(*bagFeedMasterMotor(modbusInputParameters := BagDeliverMasterMotorModbusInputs, 
                    stepsPerInchSetpoint := Globals.STEPS_PER_INCH_20_DEGREE_BAG_DELIVERY, 
                    reversePolarity := FALSE, 
                    slave := Bag_Delivery_Master_Motor);*)
bagFeedMasterMotor(ptrEIPInputs := ADR(bagDeliveryMotorInputs),
                ptrEIPOutputs := ADR(bagDeliveryMotorOutputs),
                stepsPerInchSetpoint := Globals.STEPS_PER_INCH_20_DEGREE_BAG_DELIVERY,
                //faultHandler := PRG_Bagger.faultHandler,
				reversePolarity := FALSE, 
				defaultCurrentSetpoint := 1150, 
				commFail := Bag_Delivery_EIP_Motor.eState <> IoDrvEthernetIP.AdapterState.RUNNING);
bagFeedMasterMotor.Execute();

bagFeedRearMotor(ptrEIPInputs := ADR(bagRearMotorInputs),
                ptrEIPOutputs := ADR(bagRearMotorOutputs),
                stepsPerInchSetpoint := Globals.STEPS_PER_INCH_20_DEGREE_BAG_DELIVERY,
                //faultHandler := PRG_Bagger.faultHandler,
				reversePolarity := FALSE, 
				defaultCurrentSetpoint := 1150, 
				commFail := Bag_Delivery_Rear_Motor.eState <> IoDrvEthernetIP.AdapterState.RUNNING);
bagFeedRearMotor.Execute();

IF enableONS.Q OR resetONS.Q THEN
    IF _mode = DEVICE_MODES.Manual THEN 
        state := BAG_DELIVERY_STATES.Manual;
    ELSE
        state := BAG_DELIVERY_STATES.Idle;
    END_IF
	_reset := FALSE;
	ClearCommands();
END_IF
jogForwardONS(CLK := jogForwardPB);
jogReverseONS(CLK := jogReversePB);
IF NOT enable THEN
    state := BAG_DELIVERY_STATES.Idle;
END_IF
delay();
_ready := (_mode = DEVICE_MODES.Auto) AND (NOT (state = BAG_DELIVERY_STATES.Fault) OR NOT (state = BAG_DELIVERY_STATES.Idle));

IF tensionFailONS.OSR THEN
	bagTensionFault.Trigger();
END_IF

CASE state OF
    BAG_DELIVERY_STATES.Idle :                     
													IF _mode = DEVICE_MODES.Manual THEN 
														state := BAG_DELIVERY_STATES.Manual;
													ELSIF NOT iBagNotPresent OR Globals.enableDryCycle THEN
														state := BAG_DELIVERY_STATES.Ready;
													ELSIF iBagNotPresent AND (_amFeedToEye OR _amReverseBag) THEN
														state := BAG_DELIVERY_STATES.FeedToEye;
														_amFeedToEye := FALSE;
													END_IF
													IF jogForwardONS.OSR THEN
														bagFeedMasterMotor.MoveDistance(distance := 30, 
                                                                                    acceleration := accelSetpoint, 
                                                                                    deceleration := decelSetpoint, 
                                                                                    velocity := REAL_TO_INT((1 * Globals.VELOCITY_IPS_MULTIPLIER_ELECTRIC)));
														bagFeedRearMotor.MoveDistance(distance := 30, 
                                                                                    acceleration := accelSetpoint, 
                                                                                    deceleration := decelSetpoint, 
                                                                                    velocity := REAL_TO_INT((1 * Globals.VELOCITY_IPS_MULTIPLIER_ELECTRIC)));
													ELSIF jogReverseONS.OSR THEN
														bagFeedMasterMotor.MoveDistance(distance := -30, 
                                                                                    acceleration := accelSetpoint, 
                                                                                    deceleration := decelSetpoint, 
                                                                                    velocity := REAL_TO_INT((1 * Globals.VELOCITY_IPS_MULTIPLIER_ELECTRIC)));
														bagFeedRearMotor.MoveDistance(distance := -30, 
                                                                                    acceleration := accelSetpoint, 
                                                                                    deceleration := decelSetpoint, 
                                                                                    velocity := REAL_TO_INT((1 * Globals.VELOCITY_IPS_MULTIPLIER_ELECTRIC)));
													ELSIF jogForwardONS.OSF OR jogReverseONS.OSF THEN
														bagFeedMasterMotor.Stop();
														bagFeedRearMotor.Stop();
													END_IF
    
	BAG_DELIVERY_STATES.FeedToEye :					//Feed to photoeye if not present
													bagFeedMasterMotor.MoveDistance(distance := feedToPhotoeyeSetpoint, 
                                                                                    acceleration := accelSetpoint, 
                                                                                    deceleration := decelSetpoint, 
                                                                                    velocity := REAL_TO_INT((feedToPhotoeyeSetpoint * Globals.VELOCITY_IPS_MULTIPLIER_ELECTRIC)));
													bagFeedRearMotor.MoveDistance(distance := feedToPhotoeyeSetpoint, 
                                                                                    acceleration := accelSetpoint, 
                                                                                    deceleration := decelSetpoint, 
                                                                                    velocity := REAL_TO_INT((feedToPhotoeyeSetpoint * Globals.VELOCITY_IPS_MULTIPLIER_ELECTRIC)));
													state := BAG_DELIVERY_STATES.FeedingToEye;
													
	BAG_DELIVERY_STATES.FeedingToEye :				// Stop once photoeye seen
													delay.PT := T#3S;
													delay.IN := TRUE;
													IF NOT iBagNotPresent THEN
														bagFeedMasterMotor.Stop();
														bagFeedRearMotor.Stop();
														state := BAG_DELIVERY_STATES.Idle;
														delay.IN := FALSE;
													END_IF
													IF delay.Q THEN
														state := BAG_DELIVERY_STATES.Fault;
														noBagOverEye.Trigger();
														delay.IN := FALSE;
													END_IF
	
    BAG_DELIVERY_STATES.Reverse :                    // Reverse to break perf
                                                    bagFeedMasterMotor.MoveDistance(distance := reverseDistanceSetpoint, 
                                                                                    acceleration := TO_INT((ABS(reverseDistanceSetpoint) * Globals.STEPS_PER_INCH_20_DEGREE_BAG_DELIVERY) *  accelPercent),
                                                                                    deceleration := TO_INT((ABS(reverseDistanceSetpoint) * Globals.STEPS_PER_INCH_20_DEGREE_BAG_DELIVERY) *  decelPercent), 
                                                                                    velocity := REAL_TO_INT((reverseVelocitySetpoint * Globals.VELOCITY_IPS_MULTIPLIER_ELECTRIC)));  
													bagFeedRearMotor.MoveDistance(distance := reverseDistanceSetpoint, 
                                                                                    acceleration := TO_INT((ABS(reverseDistanceSetpoint) * Globals.STEPS_PER_INCH_20_DEGREE_BAG_DELIVERY) *  accelPercent),
                                                                                    deceleration := TO_INT((ABS(reverseDistanceSetpoint) * Globals.STEPS_PER_INCH_20_DEGREE_BAG_DELIVERY) *  decelPercent), 
                                                                                    velocity := REAL_TO_INT((reverseVelocitySetpoint * Globals.VELOCITY_IPS_MULTIPLIER_ELECTRIC)));    
                                                        state := BAG_DELIVERY_STATES.Reversing;
                                                    
                                                    
    BAG_DELIVERY_STATES.Reversing :                    // Back up until we see the trailing edge of the bag
														 IF iBagNotPresent OR Globals.enableDryCycle THEN
															delay.PT := T#10MS;
															delay.IN := TRUE;
															IF delay.Q THEN
																bagFeedMasterMotor.Stop();
																bagFeedRearMotor.Stop();
																delay.IN := FALSE;
																delayForReverseFault.IN := FALSE;
																state := BAG_DELIVERY_STATES.ReverseToPrinthead;
															END_IF
														ELSIF bagFeedMasterMotor.CommandAcknowledged AND NOT iBagNotPresent THEN
															delayForReverseFault.PT := T#3000MS;
															delayForReverseFault.IN := TRUE;
															IF delayForReverseFault.Q THEN
																reverseFault.Trigger();
																bagFeedMasterMotor.Stop();
																bagFeedRearMotor.Stop();
															delayForReverseFault.IN := FALSE;
															state := BAG_DELIVERY_STATES.Fault; 
															END_IF
															
														END_IF
											
                                                  
													
	BAG_DELIVERY_STATES.ReverseToPrinthead :                    // Reverse to print head
                                                    bagFeedMasterMotor.MoveDistance(distance := reverseToPrintHeadSetpoint, 
                                                                                    acceleration := TO_INT((ABS(reverseToPrintHeadSetpoint) * Globals.STEPS_PER_INCH_20_DEGREE_BAG_DELIVERY) *  accelPercent),
                                                                                    deceleration := TO_INT((ABS(reverseToPrintHeadSetpoint) * Globals.STEPS_PER_INCH_20_DEGREE_BAG_DELIVERY) *  decelPercent), 
                                                                                    velocity := REAL_TO_INT((reverseVelocitySetpoint * Globals.VELOCITY_IPS_MULTIPLIER_ELECTRIC))); 
													bagFeedRearMotor.MoveDistance(distance := reverseToPrintHeadSetpoint, 
                                                                                    acceleration := TO_INT((ABS(reverseToPrintHeadSetpoint) * Globals.STEPS_PER_INCH_20_DEGREE_BAG_DELIVERY) *  accelPercent),
                                                                                    deceleration := TO_INT((ABS(reverseToPrintHeadSetpoint) * Globals.STEPS_PER_INCH_20_DEGREE_BAG_DELIVERY) *  decelPercent), 
                                                                                    velocity := REAL_TO_INT((reverseVelocitySetpoint * Globals.VELOCITY_IPS_MULTIPLIER_ELECTRIC)));    
                                                    state := BAG_DELIVERY_STATES.ReversingToPrintHead;
													
	BAG_DELIVERY_STATES.ReversingToPrintHead :                    // Reverse to break perf
                                                   	delay.PT := T#50MS;
													delay.IN := TRUE;
													
													IF delay.Q THEN
														IF bagFeedMasterMotor.CommandAcknowledged AND bagFeedMasterMotor.InPosition THEN
                                                        	state := BAG_DELIVERY_STATES.ReverseDone;
                                                    	END_IF
														delay.IN := FALSE;
													END_IF
                                                    
    BAG_DELIVERY_STATES.ReverseDone :                // We don't print in semi auto or manual mode.  In auto mode if the printer is selected then we move to those states
                                                    IF _mode = DEVICE_MODES.SemiAuto OR _mode = DEVICE_MODES.Manual OR (_mode  = DEVICE_MODES.Auto AND autoFeedDelay.Q) THEN
                                                        IF bagFeedMasterMotor.CommandAcknowledged THEN
															state := BAG_DELIVERY_STATES.FeedBagOut;
                                                        	remainingLength := bagLengthSetpoint;
                                                        	_amFeedBagOut := FALSE;
														END_IF
														
                                                    ELSIF (_mode  = DEVICE_MODES.Auto AND _amWaitForPrinter) THEN
                                                        IF bagFeedMasterMotor.CommandAcknowledged THEN
															state := BAG_DELIVERY_STATES.WaitingForPrinter;
															remainingLength := bagLengthSetpoint - (printLengthSetpoint + printOffsetSetpoint + printerExtraFeedLength);
															_amWaitForPrinter := FALSE;  
														END_IF  
                                                    END_IF
                                                        
                                                    
    BAG_DELIVERY_STATES.WaitingForPrinter :            // 
                                                    IF (_mode  = DEVICE_MODES.Auto AND _amPrinterReady) THEN
														IF printOffsetSetpoint <> 0 THEN
															state := BAG_DELIVERY_STATES.FeedToPrintOffset;
														ELSE
															state := BAG_DELIVERY_STATES.FedToPrintOffset;
														END_IF
                                                        
                                                        _amPrinterReady := FALSE;
                                                    END_IF
                                                        
    BAG_DELIVERY_STATES.FeedToPrintOffset :            // 
                                                    bagFeedMasterMotor.MoveDistance(distance := printOffsetSetpoint, 
                                                                                    acceleration := accelSetpoint, 
                                                                                    deceleration := decelSetpoint, 
                                                                                    velocity := REAL_TO_INT((feedVelocitySetpoint * Globals.VELOCITY_IPS_MULTIPLIER_ELECTRIC)));  
													bagFeedRearMotor.MoveDistance(distance := printOffsetSetpoint, 
                                                                                    acceleration := accelSetpoint, 
                                                                                    deceleration := decelSetpoint, 
                                                                                    velocity := REAL_TO_INT((feedVelocitySetpoint * Globals.VELOCITY_IPS_MULTIPLIER_ELECTRIC)));  
                                                        state := BAG_DELIVERY_STATES.FeedingToPrintOffset;
                                                    
    BAG_DELIVERY_STATES.FeedingToPrintOffset :        // 
													delay.PT := T#50MS;
													delay.IN := TRUE;
													
													IF delay.Q THEN
														IF bagFeedMasterMotor.CommandAcknowledged AND bagFeedMasterMotor.InPosition THEN
                                                        	state := BAG_DELIVERY_STATES.FedToPrintOffset;
                                                    	END_IF
														delay.IN := FALSE;
													END_IF
                                                    
                                                    
    BAG_DELIVERY_STATES.FedToPrintOffset :            // 
                                                    IF (_mode  = DEVICE_MODES.Auto AND _amStartPrint) THEN
                                                        state := BAG_DELIVERY_STATES.FeedAtPrintSpeed;
                                                        _amStartPrint := FALSE;
                                                    END_IF
                                                    
    BAG_DELIVERY_STATES.FeedAtPrintSpeed :            // 
													delay.PT := delayForPrintFeed;
                                                    delay.IN := TRUE;
													
													IF delay.Q THEN
														bagFeedMasterMotor.MoveDistance(distance := printLengthSetpoint + printerExtraFeedLength, 
                                                                                    acceleration := accelSetpoint, 
                                                                                    deceleration := decelSetpoint, 
                                                                                    velocity := REAL_TO_INT((printVelocitySetpoint * Globals.VELOCITY_IPS_MULTIPLIER_ELECTRIC)));  
														bagFeedRearMotor.MoveDistance(distance := printLengthSetpoint + printerExtraFeedLength, 
                                                                                    acceleration := accelSetpoint, 
                                                                                    deceleration := decelSetpoint, 
                                                                                    velocity := REAL_TO_INT((printVelocitySetpoint * Globals.VELOCITY_IPS_MULTIPLIER_ELECTRIC)));  
                                                        state := BAG_DELIVERY_STATES.FeedingAtPrintSpeed;
														delay.IN := FALSE;
													END_IF
                                                    
    BAG_DELIVERY_STATES.FeedingAtPrintSpeed :        // 
													delay.PT := T#50MS;
													delay.IN := TRUE;
													IF delay.Q THEN
														IF bagFeedMasterMotor.CommandAcknowledged AND bagFeedMasterMotor.InPosition THEN
                                                        	state := BAG_DELIVERY_STATES.FedAtPrintSpeed;
                                                    	END_IF
														delay.IN := FALSE;
													END_IF
                                                   
                                                    
    BAG_DELIVERY_STATES.FedAtPrintSpeed :            // 
                                                    IF (_mode  = DEVICE_MODES.Auto AND _amPrinterDone) THEN
                                                        state := BAG_DELIVERY_STATES.FeedBagOut;
                                                        _amPrinterDone := FALSE;
                                                    END_IF
                                                    
    BAG_DELIVERY_STATES.FeedBagOut :                // Feed bag length out
                                                    //bagFeedMasterMotor.MoveDistanceFinal(distance := (remainingLength + sealOffsetSetpoint + (reverseToPrintHeadSetpoint*-1)), 
													bagFeedMasterMotor.MoveDistanceFinal(distance := (remainingLength + sealBarToPrintHeadLength) - sealOffsetSetpoint, 
                                                                                        acceleration := accelSetpoint, 
                                                                                        deceleration := decelSetpoint, 
                                                                                        velocity := REAL_TO_INT((feedVelocitySetpoint * Globals.VELOCITY_IPS_MULTIPLIER_ELECTRIC)));
													bagFeedRearMotor.MoveDistance(distance := (remainingLength + sealBarToPrintHeadLength) - sealOffsetSetpoint, 
                                                                                        acceleration := accelSetpoint, 
                                                                                        deceleration := decelSetpoint, 
                                                                                        velocity := REAL_TO_INT((feedVelocitySetpoint * Globals.VELOCITY_IPS_MULTIPLIER_ELECTRIC)));
                                                    state := BAG_DELIVERY_STATES.FeedingBagOut;    
    
    BAG_DELIVERY_STATES.FeedingBagOut :                // Wait until move is done
													delay.PT := T#50MS;
													delay.IN := TRUE;
													IF delay.Q THEN
														IF bagFeedMasterMotor.CommandAcknowledged AND bagFeedMasterMotor.InPosition THEN
                                                        state := BAG_DELIVERY_STATES.FedBagOut;
														
                                                    	END_IF
														delay.IN := FALSE;
													END_IF
                                                    
    
    BAG_DELIVERY_STATES.FedBagOut :                    // Go to the next ready state
                                                    IF _mode = DEVICE_MODES.Manual THEN 
                                                        state := BAG_DELIVERY_STATES.Manual;
                                                    ELSE
                                                        state := BAG_DELIVERY_STATES.Ready;
                                                    END_IF
													HMIData.driveRollerClean.SetCount(HMIData.driveRollerClean.count + TO_INT(bagLengthSetpoint));
                                                    Globals.bagDeliveryCycleCount := Globals.bagDeliveryCycleCount + 1;
    
    BAG_DELIVERY_STATES.Ready :                        IF (_mode = DEVICE_MODES.Auto AND _amReverseBag) OR _mode = DEVICE_MODES.SemiAuto THEN 
                                                        state := BAG_DELIVERY_STATES.Reverse;
                                                        ClearCommands();
                                                    END_IF 
													_amFeedToEye := FALSE;
													IF iBagNotPresent AND NOT Globals.enableDryCycle THEN 
														state := BAG_DELIVERY_STATES.Idle;
													END_IF
													IF jogForwardONS.OSR THEN
														bagFeedMasterMotor.MoveDistance(distance := 30, 
                                                                                    acceleration := accelSetpoint, 
                                                                                    deceleration := decelSetpoint, 
                                                                                    velocity := REAL_TO_INT((1 * Globals.VELOCITY_IPS_MULTIPLIER_ELECTRIC)));
														bagFeedRearMotor.MoveDistance(distance := 30, 
                                                                                    acceleration := accelSetpoint, 
                                                                                    deceleration := decelSetpoint, 
                                                                                    velocity := REAL_TO_INT((1 * Globals.VELOCITY_IPS_MULTIPLIER_ELECTRIC)));
													ELSIF jogReverseONS.OSR THEN
														bagFeedMasterMotor.MoveDistance(distance := -30, 
                                                                                    acceleration := accelSetpoint, 
                                                                                    deceleration := decelSetpoint, 
                                                                                    velocity := REAL_TO_INT((1 * Globals.VELOCITY_IPS_MULTIPLIER_ELECTRIC)));
														bagFeedRearMotor.MoveDistance(distance := -30, 
                                                                                    acceleration := accelSetpoint, 
                                                                                    deceleration := decelSetpoint, 
                                                                                    velocity := REAL_TO_INT((1 * Globals.VELOCITY_IPS_MULTIPLIER_ELECTRIC)));
													ELSIF jogForwardONS.OSF OR jogReverseONS.OSF THEN
														bagFeedMasterMotor.Stop();
														bagFeedRearMotor.Stop();
													END_IF
    
    BAG_DELIVERY_STATES.Fault :                        ClearCommands();
													IF jogForwardONS.OSR THEN
														bagFeedMasterMotor.MoveDistance(distance := 30, 
                                                                                    acceleration := accelSetpoint, 
                                                                                    deceleration := decelSetpoint, 
                                                                                    velocity := REAL_TO_INT((1 * Globals.VELOCITY_IPS_MULTIPLIER_ELECTRIC)));
													ELSIF jogReverseONS.OSR THEN
														bagFeedMasterMotor.MoveDistance(distance := -30, 
                                                                                    acceleration := accelSetpoint, 
                                                                                    deceleration := decelSetpoint, 
                                                                                    velocity := REAL_TO_INT((1 * Globals.VELOCITY_IPS_MULTIPLIER_ELECTRIC)));
													ELSIF jogForwardONS.OSF OR jogReverseONS.OSF THEN
														bagFeedMasterMotor.Stop();
														bagFeedRearMotor.Stop();
													END_IF
    
    BAG_DELIVERY_STATES.Manual :                    IF _mode = DEVICE_MODES.Auto THEN
														state := BAG_DELIVERY_STATES.Ready;	
													END_IF
													// Manually feed bags out
                                                    IF feedBagPB THEN
                                                        state := BAG_DELIVERY_STATES.Reverse;
                                                        feedBagPB := FALSE;
                                                    END_IF
                                                        
END_CASE

END_FUNCTION_BLOCK

// FBs/Unused/ElectricPressureBarFB
FUNCTION_BLOCK ElectricPressureBarFB IMPLEMENTS IComponentStatus
VAR_INPUT
    enable : BOOL;
END_VAR
VAR_IN_OUT

END_VAR
VAR_OUTPUT
END_VAR
VAR
    electricPressureBarMotor : FB_FestoMotor();
    delay: TON := (PT := T#1S);
    state : PRESSURE_BAR_STATES;
    enableElectricPressureBarONS : R_TRIG();
    
    _mode : DEVICE_MODES;    // Auto-SemiAuto-Manual
    _ready : BOOL;            // Ready to be controlled
    _amOpenJaw : BOOL;    // Auto Mode Open Jaw Command
    _amCloseJaw : BOOL;     // Auto Mode Close Jaw Command
END_VAR

//    Function Block: ElectricPressureBarFB
//    Description: This function block is the state machine for the electric pressure bar
//    
//    Created by: Ben Hess
//    Created Date: Monday, April 16, 2018

electricPressureBarMotor(deviceType := FML.CMMP_AS,
                                        isFPCActive := TRUE, 
                                        ptrReadFHPPRegister := ADR(%IW145), 
                                        ptrReadFPCRegister := ADR(%IW149),
                                        ptrWriteFHPPRegister := ADR(%QW82),
                                        ptrWriteFPCRegister := ADR(%QW86));                                    
electricPressureBarMotor.Execute();

delay();

//Report as ready if mode is auto and we're not faulted
_ready := (_mode = DEVICE_MODES.Auto) AND NOT (state = PRESSURE_BAR_STATES.Fault);


enableElectricPressureBarONS(CLK := enable);
IF enableElectricPressureBarONS.Q THEN
    state := PRESSURE_BAR_STATES.Idle;
END_IF

IF NOT enable THEN
        state := PRESSURE_BAR_STATES.Fault;
END_IF

CASE state OF
    PRESSURE_BAR_STATES.Idle:        IF enable AND _mode = DEVICE_MODES.SemiAuto OR (_mode = DEVICE_MODES.Auto AND _amCloseJaw) THEN
                                        state := PRESSURE_BAR_STATES.CloseJaw;
                                        _amCloseJaw := FALSE;
                                    END_IF
    
    PRESSURE_BAR_STATES.OpenJaw:    electricPressureBarMotor.ExecuteStoredProgram(1);
                                    IF electricPressureBarMotor.CommandAcknowledged THEN
                                        state := PRESSURE_BAR_STATES.OpeningJaw;
                                        Globals.electricPressureBarCount := Globals.electricPressureBarCount + 1;
                                    END_IF
        
    
    PRESSURE_BAR_STATES.OpeningJaw:    
                                    IF electricPressureBarMotor.ActiveStoredProgramNumber = 1 AND electricPressureBarMotor.InPosition THEN
                                        state := PRESSURE_BAR_STATES.JawOpened;
                                    END_IF
                                    
    PRESSURE_BAR_STATES.JawOpened:     IF _mode = DEVICE_MODES.SemiAuto THEN
                                        delay.IN := TRUE;
                                        IF delay.Q THEN
                                            state := PRESSURE_BAR_STATES.CloseJaw;
                                            delay.IN := FALSE;
                                        END_IF
                                    ELSIF _mode = DEVICE_MODES.Auto AND _amCloseJaw THEN
                                        state := PRESSURE_BAR_STATES.CloseJaw;
                                        _amCloseJaw := FALSE;
                                    END_IF
        
    PRESSURE_BAR_STATES.CloseJaw:    electricPressureBarMotor.ExecuteStoredProgram(2);
                                    IF electricPressureBarMotor.CommandAcknowledged THEN
                                        state := PRESSURE_BAR_STATES.ClosingJaw;
                                        Globals.electricPressureBarCount := Globals.electricPressureBarCount + 1;
                                    END_IF
                                    
    
    PRESSURE_BAR_STATES.ClosingJaw:    IF electricPressureBarMotor.ActiveStoredProgramNumber = 2 AND electricPressureBarMotor.InPosition THEN
                                        state := PRESSURE_BAR_STATES.JawClosed;
                                    END_IF
                                    
    PRESSURE_BAR_STATES.JawClosed:    IF _mode = DEVICE_MODES.SemiAuto THEN
                                        delay.IN := TRUE;
                                        IF delay.Q THEN
                                            state := PRESSURE_BAR_STATES.OpenJaw;
                                            delay.IN := FALSE;
                                        END_IF
                                    ELSIF _mode = DEVICE_MODES.Auto AND _amOpenJaw THEN
                                        state := PRESSURE_BAR_STATES.OpenJaw;
                                        _amOpenJaw := FALSE;
                                    END_IF
    
    PRESSURE_BAR_STATES.Fault:        ClearCommands();        
    
    
END_CASE

END_FUNCTION_BLOCK

// FBs/Unused/MotorizedSealFlattenersFB
FUNCTION_BLOCK MotorizedSealFlattenersFB EXTENDS BaseComponentFB IMPLEMENTS IComponentStatus
VAR_INPUT
    {warning 'TODO: Make a struct for some of these - too many inputs'}
	sealFlattenersVerticalAxis : ICylinder();
    clearanceOffset : REAL := 0.75;        // Clearance Offset in inches
    inSetpoint : REAL := 1.25;            // In setpoint in inches
    outSetpoint : REAL := 17.7;            // Out (sealing) setpoint in inches
    bagHoldingSetpoint : REAL := 17;    // Bag holding setpoint in inches            
    clearanceSpeed : INT := 3000;        // Speed to move in clearance move
    moveInSpeed : INT := 3000;            // Speed to move in in move
    moveOutSpeed : INT := 1000;            // Speed to move in out move
    moveBagHoldingSpeed : INT := 10000;    // Speed to move in bag holding move
    fingersUpSetpoint : REAL := 0;     // Fingers Up setpoint in inches
    fingersDownSetpoint : REAL := 1.1; // Fingers down setpoint in inches
    moveFingersSpeed : INT := 2000;        // Speed to move fingers
    horizontalAxisAccel : INT := 1000;    // Accel setpoint for horizontal axis
    horizontalAxisDecel : INT := 1000;    // Decel Setpoint for horizontal axis
    verticalAxisAccel : INT := 150;    // Accel setpoint for vertical axis
    verticalAxisDecel : INT := 150;    // Decel Setpoint for vertical axis
    testMovePB : BOOL;
    testMoveSP : REAL;
    stopPB : BOOL;
    startPB : BOOL;
    nextSeqPB : BOOL;
    delay : TON := (PT:= T#300MS);
	fingersDownDelay : Standard.TON := (PT := T#200MS);
	
	manualPosSetpoint : REAL;
	
END_VAR
VAR_IN_OUT
	jogIn : BOOL;
	jogOut : BOOL;
	raiseService : BOOL;
	lowerService : BOOL;
	moveToManualSetpoint : BOOL;
END_VAR
VAR_OUTPUT
    state : SEAL_FLATTENER_STATES;
END_VAR
VAR
    //pressureBarMotor : FB_FestoMotor();
    //sealFlattenersVerticalAxisMotor : FB_AppliedMotionStepServoRTU();
	jogInONS: FB_ONS;
	jogOutONS: FB_ONS;
	jogSpeed : INT := 100;
    sealFlattenersHorizontalAxisMotor : FB_AppliedMotionStepServoEIPBaseQX();
	defaultCurrentMSF : DINT := 150;
	outCurrentMSF : DINT := 150;
	bagHoldingCurrentMSF : DINT := 85;
    enableMotorizedSealFlattenersONS : R_TRIG();    
    _amMoveOut : BOOL;                // Auto mode move out command
	_amMoveIn : BOOL;
    _amMoveClearance : BOOL;            // Auto mode move Clearance command
    _amMoveInToBagHolding : BOOL;    // Auto mode move in then bag holding command
END_VAR

//    Function Block:  MotorizedSealFlattenersFB
//    Description: State machine and motor management for motorized seal flateners
//    Currently, this code requires one to use the Oriental drive with pre-programmed 
//    sequence for the horizontal axis
//    Created by: Ben Hess
//    Created Date: Friday, April 6, 2018
SUPER^();
// Setup and execute 2 motor axis'

// Temporary delay between states for testing
fingersDownDelay();
delay();
jogInONS(CLK := jogIn);
jogOutONS(CLK := jogOut);
IF autoModeSelected THEN
    delay.PT := T#300MS;
ELSE
    delay.PT := T#750MS;
END_IF

outSetpoint := HMIData.bagWidth + 0.2;
bagHoldingSetpoint := HMIData.bagWidth;

// Setup the vertical axis motor
sealFlattenersVerticalAxis.Execute();

// Setup the horizontal axis motor 
(*
sealFlattenersHorizontalAxisMotor(modbusInBuffer := OrientalMotorModbusRead,
                stepsPerInchSetpoint := 125,
                reversePolarity := FALSE,
                operatingCurrentDefault := 500,
                modbusCommandOutBuffer := OrientalMotorCommandWrites,
                modbusParametersOutBuffer := OrientalMotorParameterWrites,
                triggerCommandWrite => OrientalMotorTriggerCommandWrite,
                triggerParameterWrite => OrientalMotorTriggerParameterWrite);                
sealFlattenersHorizontalAxisMotor.Execute();
*)

sealFlattenersHorizontalAxisMotor(ptrEIPInputs := ADR(sealFlattenerHorizontalMotorInputs),
                ptrEIPOutputs := ADR(sealFlattenerHorizontalMotorOutputs),
                stepsPerInchSetpoint := Globals.STEPS_PER_INCH_SEAL_FLATTENER_HORIZONTAL_AXIS_MOTOR,
                faultHandler := PRG_Bagger.faultHandler,
				reversePolarity := TRUE, 
				defaultCurrentSetpoint := defaultCurrentMSF, 
				commFail := MSFMotor.eState <> IoDrvEthernetIP.AdapterState.RUNNING,
				isHomable := TRUE);
				
sealFlattenersHorizontalAxisMotor.Execute();

//Report as ready if mode is auto and we're not faulted
_ready := (_mode = DEVICE_MODES.Auto) AND NOT (state = SEAL_FLATTENER_STATES.Fault);

enableMotorizedSealFlattenersONS(CLK := enable);
IF stopPB THEN
    sealFlattenersHorizontalAxisMotor.Stop();
    stopPB := FALSE;
END_IF

IF startPB AND semiAutoModeSelected THEN 
    //sealFlattenersHorizontalAxisMotor.StartOperation();
    startPB := FALSE;
END_IF

IF nextSeqPB THEN 
    //sealFlattenersHorizontalAxisMotor.NextSequence();
    nextSeqPB := FALSE;
END_IF

IF testMovePB THEN
    sealFlattenersHorizontalAxisMotor.MoveToPosition(position := (testMoveSP), acceleration := 100, deceleration := 100, velocity := 600);
    testMovePB := FALSE;
END_IF

IF enableONS.Q OR resetONS.Q THEN 
    state := SEAL_FLATTENER_STATES.Idle;
	sealFlattenersHorizontalAxisMotor.Reset();
	_reset := FALSE;
	ClearCommands();
END_IF

IF NOT enable THEN
    state := SEAL_FLATTENER_STATES.Fault;
END_IF

// State amchine for motorized seal flatteners
CASE state OF
    

    SEAL_FLATTENER_STATES.Idle :                                    //If enabled move to out
                                                                    IF enable AND semiAutoModeSelected OR (autoModeSelected AND _amMoveOut) THEN
                                                                        state := SEAL_FLATTENER_STATES.MoveFlattenersOut;
                                                                        ClearCommands();
                                                                    END_IF
																	
																	IF enable AND autoModeSelected AND _amMoveIn OR _amMoveInToBagHolding THEN
																	//IF enable AND autoModeSelected AND _amMoveIn THEN
																		sealFlattenersVerticalAxis.Retract();
																		state := SEAL_FLATTENER_STATES.MoveFlattenersIn;
																		ClearCommands();
																	END_IF
																	
																	IF jogInONS.OSR THEN
																		sealFlattenersHorizontalAxisMotor.MoveDistance(distance := -18, 
																									acceleration := horizontalAxisAccel, 
																									deceleration := horizontalAxisDecel, 
																									velocity := jogSpeed);
																	ELSIF jogOutONS.OSR THEN
																		sealFlattenersHorizontalAxisMotor.MoveDistance(distance := 18, 
																									acceleration := horizontalAxisAccel, 
																									deceleration := horizontalAxisDecel, 
																									velocity := jogSpeed);
																	ELSIF jogInONS.OSF OR jogOutONS.OSF THEN
																		sealFlattenersHorizontalAxisMotor.Stop();
																	END_IF
																	
																	IF raiseService THEN
																		sealFlattenersVerticalAxis.Retract();  
																		raiseService := FALSE;
																	ELSIF lowerService THEN
																		sealFlattenersVerticalAxis.Extend();  
																		lowerService := FALSE;
																	END_IF
																	
																	IF moveToManualSetpoint THEN
																		sealFlattenersHorizontalAxisMotor.MoveToPosition(position := manualPosSetpoint, 
																									acceleration := horizontalAxisAccel, 
																									deceleration := horizontalAxisDecel, 
																									velocity := moveFingersSpeed);
																		moveToManualSetpoint := FALSE;
																	END_IF
																	
                                                                    
    SEAL_FLATTENER_STATES.MoveFlattenersOut :                        // Move flatteners to out position
                                                                
                                                                    //sealFlattenersHorizontalAxisMotor.StartOperation();
                                                                    sealFlattenersHorizontalAxisMotor.MoveToPositionTorque(position := outSetpoint, 
                                                                                                                        acceleration := horizontalAxisAccel,
                                                                                                                        deceleration := horizontalAxisDecel,
                                                                                                                        velocity := moveOutSpeed,
																														current := outCurrentMSF);                                                    
                                                                    state := SEAL_FLATTENER_STATES.MovingFlattenersOut;
                                                                    
                                                                    
    SEAL_FLATTENER_STATES.MovingFlattenersOut :                        // 
                                                                    delay.IN := TRUE;
                                                                    IF delay.Q THEN
																		IF sealFlattenersHorizontalAxisMotor.CommandAcknowledged AND sealFlattenersHorizontalAxisMotor.CurrentPosition >= (bagHoldingSetpoint - 1.5) THEN
																			state := SEAL_FLATTENER_STATES.MovedFlattenersOut;
                                                                        	delay.IN := FALSE; 
																		END_IF
                                                                    END_IF
                                                                    
    SEAL_FLATTENER_STATES.MovedFlattenersOut :                        // Move flatteners to clearance position state
                                                                    IF enable AND semiAutoModeSelected OR (autoModeSelected AND _amMoveClearance) THEN
                                                                        state := SEAL_FLATTENER_STATES.MoveFlattenersUpAndToClearance;
                                                                        ClearCommands();
                                                                    END_IF
    
    
    SEAL_FLATTENER_STATES.MoveFlattenersUpAndToClearance :                // Move flatteners to clearance position
                                                                    
                                                                    //sealFlattenersHorizontalAxisMotor.NextSequence();
                                                                    sealFlattenersHorizontalAxisMotor.MoveToPosition(position := (outSetpoint - clearanceOffset), 
                                                                                                                        acceleration := horizontalAxisAccel,
                                                                                                                        deceleration := horizontalAxisDecel,
                                                                                                                        velocity := moveOutSpeed);    
                                                                   	sealFlattenersVerticalAxis.Retract();                                                       
                                                                    state := SEAL_FLATTENER_STATES.MovingFlattenersUpAndToClearance;    
    
    
    
    SEAL_FLATTENER_STATES.MovingFlattenersUpAndToClearance :        delay.IN := TRUE;
                                                                    IF delay.Q THEN
																		IF sealFlattenersHorizontalAxisMotor.CommandAcknowledged AND sealFlattenersHorizontalAxisMotor.InPosition THEN
																			state := SEAL_FLATTENER_STATES.MovedFlattenersUpAndToClearance;    
                                                                        	delay.IN := FALSE;
																		END_IF
                                                                    END_IF
                                                                    
                                                                    
    SEAL_FLATTENER_STATES.MovedFlattenersUpAndToClearance :                // Move flatteners to up state
                                                                    IF enable AND semiAutoModeSelected OR (autoModeSelected AND (_amMoveInToBagHolding OR _amMoveIn)) THEN
                                                                        state := SEAL_FLATTENER_STATES.MoveFlattenersIn;
                                                                        //ClearCommands();
                                                                    END_IF
                                        
                                                                    
    SEAL_FLATTENER_STATES.MoveFlattenersIn :                        // Move flatteners up and in
                                                                    //sealFlattenersHorizontalAxisMotor.NextSequence();    
                                                                    sealFlattenersHorizontalAxisMotor.MoveToPosition(position := inSetpoint, 
                                                                                                                        acceleration := horizontalAxisAccel,
                                                                                                                        deceleration := horizontalAxisDecel,
                                                                                                                        velocity := moveInSpeed);                                                    
                                                                    state := SEAL_FLATTENER_STATES.MovingFlattenersIn;
                                                                    
                                                                    
    SEAL_FLATTENER_STATES.MovingFlattenersIn :                        // If we did that command well move on 
                                                                        delay.IN := TRUE;
                                                                        IF delay.Q THEN
																			IF sealFlattenersHorizontalAxisMotor.CommandAcknowledged AND sealFlattenersHorizontalAxisMotor.InPosition THEN
																				state := SEAL_FLATTENER_STATES.MovedFlattenersIn;
                                                                           		delay.IN := FALSE;    
																			END_IF
                                                                        END_IF 
                                                                    
    SEAL_FLATTENER_STATES.MovedFlattenersIn :                        // Now that we're up and in move to down and 4 corners/bag holding
                                                                    IF enable AND semiAutoModeSelected OR (autoModeSelected AND _amMoveInToBagHolding) THEN
                                                                        state := SEAL_FLATTENER_STATES.MoveFlattenersDown;
                                                                        ClearCommands();
                                                                    END_IF    
    
    SEAL_FLATTENER_STATES.MoveFlattenersDown :            // Do moves for down and bag holding
                                                                        
                                                                        sealFlattenersVerticalAxis.Extend();
                                                                                                                                                                                
                                                                        state := SEAL_FLATTENER_STATES.MovingFlattenersDown;
                                                                        
    SEAL_FLATTENER_STATES.MovingFlattenersDown :            
                                                                        //IF sealFlattenersVerticalAxis.CommandAcknowledged AND sealFlattenersVerticalAxis.InPosition THEN
                                                                       	fingersDownDelay.IN := TRUE;
																	  	IF fingersDownDelay.Q THEN
																			state := SEAL_FLATTENER_STATES.MovedFlattenersDown;
																			fingersDownDelay.IN := FALSE;
																		END_IF 
																		
                                                                        //END_IF 
                                                                        
    SEAL_FLATTENER_STATES.MovedFlattenersDown :            state := SEAL_FLATTENER_STATES.MoveFlattenersToBagHolding;
                                                                    
                                                                    
    SEAL_FLATTENER_STATES.MoveFlattenersToBagHolding :            // Do moves for down and bag holding
                                                                        //sealFlattenersHorizontalAxisMotor.NextSequence();    
                                                                        sealFlattenersHorizontalAxisMotor.MoveToPositionTorque(position := bagHoldingSetpoint, 
                                                                                                                        acceleration := horizontalAxisAccel,
                                                                                                                        deceleration := horizontalAxisDecel,
                                                                                                                        velocity := moveBagHoldingSpeed,
																														current := bagHoldingCurrentMSF);                                                
                                                                        state := SEAL_FLATTENER_STATES.MovingFlattenersToBagHolding;
                                                                        
    SEAL_FLATTENER_STATES.MovingFlattenersToBagHolding :            delay.IN := TRUE;
                                                                        IF delay.Q THEN
																			IF sealFlattenersHorizontalAxisMotor.CommandAcknowledged THEN
																				state := SEAL_FLATTENER_STATES.MovedFlattenersToBagHolding;
                                                                            	delay.IN := FALSE; 
																			END_IF   
                                                                        END_IF 
                                                                        
    SEAL_FLATTENER_STATES.MovedFlattenersToBagHolding :            state := SEAL_FLATTENER_STATES.Idle;
																		HMIData.motorizedSealFlattenerCycles.Increment();
                                                                        Globals.motorizedSealFlattenersCount := Globals.motorizedSealFlattenersCount +1;
                                                                        Globals.sealFlattenerFingersCount := Globals.sealFlattenerFingersCount +1;
    SEAL_FLATTENER_STATES.Ready :
    SEAL_FLATTENER_STATES.Fault :
END_CASE

END_FUNCTION_BLOCK

// FBs/Unused/PickAndPlaceFB
FUNCTION_BLOCK PickAndPlaceFB EXTENDS BaseComponentFB
VAR_INPUT
	XAxisMotor : IPositionableMotor;	// X Axis Motor
	YAxisMotor : IPositionableMotor;	// Y Axis Motor
	ZAxisMotor : IPositionableMotor;	// Z Axis Motor
END_VAR
VAR_OUTPUT
	state : VACUUM_PICKER_STATES;	 //State indication
END_VAR
VAR
	
	accel : INT := 2000;
	decel : INT := 2000;
	velo : INT := 2000;
	zVelo : INT := 12000;
END_VAR

//	Function Block: PickAndPlaceFB
//	Description: This provides the methods and state machine to operate the Vacuum Head pick and place machine
//	
//	Created by: Ben Hess
//	Created Date: Friday, June 1, 2018

// Run the base FB
SUPER^();

// Set up the 3 motors.

// X Axis moves out and in relative to the machine. Out is 0in, max in is 7.5in.


IF enableONS.Q THEN
    IF _mode = DEVICE_MODES.Manual THEN 
        state := VACUUM_PICKER_STATES.Manual;
    ELSE
        state := VACUUM_PICKER_STATES.Ready;
    END_IF
END_IF

IF NOT enable THEN
    state := VACUUM_PICKER_STATES.Idle;
END_IF

_ready := (_mode = DEVICE_MODES.Auto) AND NOT (state = VACUUM_PICKER_STATES.Fault);


CASE state OF
	VACUUM_PICKER_STATES.Idle :
	VACUUM_PICKER_STATES.Home :								// Move everything to home position
															XAxisMotor.MoveToPosition(6, accel,decel,velo);
															YAxisMotor.MoveToPosition(15, accel,decel,velo);
															ZAxisMotor.MoveToPosition(1, accel,decel,zVelo);
															state := VACUUM_PICKER_STATES.Homing;
															
	VACUUM_PICKER_STATES.Homing :							// Move on if all motors report ready
															IF XAxisMotor.CurrentPosition = 6
																AND YAxisMotor.CurrentPosition = 15
																AND ZAxisMotor.CurrentPosition = 1 THEN
																	state := VACUUM_PICKER_STATES.Homed;
															END_IF
															
	VACUUM_PICKER_STATES.Homed :							// 
															state :=VACUUM_PICKER_STATES.XAxisMoveIn;
															
	VACUUM_PICKER_STATES.XAxisMoveIn :						// Move XAxis in 
															XAxisMotor.MoveToPosition(0,accel,decel,velo);
															state := VACUUM_PICKER_STATES.XAxisMovingIn;
															
	VACUUM_PICKER_STATES.XAxisMovingIn :					// 
															IF XAxisMotor.CurrentPosition = 0 THEN
																state := VACUUM_PICKER_STATES.XaxisMovedIn;
															END_IF
															
	VACUUM_PICKER_STATES.XaxisMovedIn :						// 
															state := VACUUM_PICKER_STATES.VacuumTurnOn;
															
	VACUUM_PICKER_STATES.VacuumTurnOn :						// 
															state := VACUUM_PICKER_STATES.VacuumHeadDown;
															
	VACUUM_PICKER_STATES.VacuumHeadDown :					// 
															ZAxisMotor.MoveToPosition(150,accel,decel,zVelo);
															state := VACUUM_PICKER_STATES.YAxisMoveDown;
															
	VACUUM_PICKER_STATES.YAxisMoveDown :					// 
															YAxisMotor.MoveToPosition(1,accel,decel,velo);
															state := VACUUM_PICKER_STATES.VacuumHeadAndYAxisMovingDown;
															
	VACUUM_PICKER_STATES.VacuumHeadAndYAxisMovingDown :		// 
															IF YAxisMotor.CurrentPosition = 1
																AND ZAxisMotor.CurrentPosition = 150 THEN
																state := VACUUM_PICKER_STATES.VacuumHeadAndYAxisMovedDown;  
															END_IF	
															
	VACUUM_PICKER_STATES.VacuumHeadAndYAxisMovedDown :		// 
															state := VACUUM_PICKER_STATES.VacuumTurnOff;
															
	VACUUM_PICKER_STATES.VacuumTurnOff :					// 
															state := VACUUM_PICKER_STATES.ConveyorTurnOn;
															
	VACUUM_PICKER_STATES.ConveyorTurnOn :					// 
															state := VACUUM_PICKER_STATES.ConveyorMoving;
															
	VACUUM_PICKER_STATES.ConveyorMoving :					// 
															state := VACUUM_PICKER_STATES.ConveyorDone;
															
	VACUUM_PICKER_STATES.ConveyorDone :						// 
															state := VACUUM_PICKER_STATES.Ready;
															
	VACUUM_PICKER_STATES.Fault :							// 
																													
	
	VACUUM_PICKER_STATES.Ready :							IF semiAutoModeSelected THEN
																state := VACUUM_PICKER_STATES.Home;
															END_IF
	VACUUM_PICKER_STATES.Manual :
END_CASE

END_FUNCTION_BLOCK

// FBs/Unused/PrinterFB
FUNCTION_BLOCK PrinterFB EXTENDS BaseComponentFB IMPLEMENTS IComponentStatus
VAR_INPUT
    autoSendLabel :BOOL;    // Automatically send a label                
END_VAR
VAR_OUTPUT
    state : PRINTER_STATES;         // Printer State Machine
	oLowerPrintHead : BOOL;
	printHeadDebounced : BOOL;
	
END_VAR
VAR
    _amPrintNow : BOOL;                // Auto mode - print now
    _amSendPrintSignal : BOOL;        // Auto mode - send print signal
    _amGoToIdle : BOOL;                // Auto mode - Acked, go back to idle mode
    printHeadDebounce : TON;
    printHeadDebouneSetpoint : TIME := T#50MS;
    tcpServer : FB_TCPClient();
END_VAR

VAR_IN_OUT
END_VAR

//    Function Block: Printer
//    Description: This program manages the aspects of a (Zebra) printer
//    Created by: Ben Hess
//    Created Date: April 2nd, 2018
SUPER^();
// Enable TCP Server for label sending
tcpServer();

//Report as ready if mode is auto and we're not faulted
_ready := (_mode = DEVICE_MODES.Auto) AND NOT (state = PRINTER_STATES.Fault);

printHeadDebounce(PT:= printHeadDebouneSetpoint, Q=> printHeadDebounced);
IF enableONS.Q OR resetONS.Q THEN
    state := PRINTER_STATES.Idle;
	_reset := FALSE;
	_amGoToIdle := FALSE;
	_amSendPrintSignal := FALSE;
	_amPrintNow := FALSE;
END_IF

IF NOT enable THEN
    state := PRINTER_STATES.Fault;
	oRunPrinterRibbonUnwindMotor := FALSE;
	oLowerPrintHead := FALSE;
END_IF



//State machine for the printer
CASE state OF
    PRINTER_STATES.Idle :                            //Go to waiting for data if printer is ready
                                                    oRunPrinterRibbonUnwindMotor := FALSE;
													oPrinterStartPrint := FALSE;
													oLowerPrintHead := FALSE;
													printHeadDebounce.IN := FALSE;
													IF NOT printerDataReady THEN
                                                        IF autoSendLabel THEN
                                                            tcpServer.SendLabel();
                                                        END_IF
                                                        state := PRINTER_STATES.WaitingForData;
                                                    ELSE
                                                        state := PRINTER_STATES.DataReady;
                                                    END_IF
                                                    
                                        
    
    PRINTER_STATES.WaitingForData :                    //If printerDataReady drops out the label data was received
                                                    
                                                    IF printerDataReady THEN
                                                        state := PRINTER_STATES.DataReady;    
                                                    END_IF
                                                
    PRINTER_STATES.DataReady :                        // Wait for command to begin printing
                                                    IF NOT printerDataReady THEN
														state := PRINTER_STATES.Idle;
													END_IF
													IF _mode = DEVICE_MODES.Auto AND _amPrintNow THEN
                                                        state := PRINTER_STATES.BeginPrintCycle;
                                                        _amPrintNow := FALSE;
                                                        oLowerPrintHead := TRUE;
                                                        oRunPrinterRibbonUnwindMotor := TRUE;
														//oPrinterStartPrint := TRUE;
                                                    END_IF                                    
            
    
    PRINTER_STATES.BeginPrintCycle :                // Start printing
                                                    
                                                    printHeadDebounce.IN := TRUE;
                                                    IF printHeadDebounce.Q AND _amSendPrintSignal THEN
                                                        oPrinterStartPrint := TRUE;
                                                        state := PRINTER_STATES.Printing;
                                                        printHeadDebounce.IN := FALSE;
                                                        _amSendPrintSignal := FALSE;
                                                    END_IF                                                    
                                        
    
    PRINTER_STATES.FeedAtPrintSpeed :                //

                                                    
                                                                                                
                                        
    PRINTER_STATES.Printing :                        //While printing, wait for End of Print signal
                                                    IF printerEndOfPrint THEN
                                                        oPrinterStartPrint := FALSE;
                                                        oLowerPrintHead := FALSE;
                                                        
                                                        state := PRINTER_STATES.DonePrinting;    
                                                    END_IF
                                        
    PRINTER_STATES.DonePrinting :                    //Done printing, feed a little more through
                                                    IF _mode = DEVICE_MODES.Auto AND _amGoToIdle THEN
                                                        oRunPrinterRibbonUnwindMotor := FALSE;
                                                        state := PRINTER_STATES.Idle;
                                                        _amGoToIdle := FALSE;
														HMIData.printerCycles.Increment();
														HMIData.printHeadClean.Increment();
                                                        Globals.printerCycleCounts := Globals.printerCycleCounts + 1;
                                                    END_IF
        
    PRINTER_STATES.FeedThrough :                        
                                        
    PRINTER_STATES.Ready :                        
                                        
    PRINTER_STATES.Fault :                        
                                        
END_CASE

END_FUNCTION_BLOCK

// Function Blocks/Diagnostics/FB_StateRateTracking
FUNCTION_BLOCK FB_StateRateTracking
VAR CONSTANT
	NbMaxArrayDepth: INT := 30;
	stopTime: TIME := T#30S;
END_VAR

VAR_INPUT
	stateName : string;
	cntUp: BOOL;
	state:INT;
	trackingEnable: BOOL;
END_VAR
VAR_OUTPUT
END_VAR
VAR
	cntUpONS: R_TRIG;
	stateTimer:TON;
	laststate: INT;
	count_index :INT :=0;
	clr:BOOL:=FALSE;
	speedTracking : ARRAY[0..NbMaxArrayDepth] OF stateRateKeyPair;
	speedTracking_mt : ARRAY[0..20] OF time := [21(T#0MS)]; 
	state_index : INT:=0;
	index: INT;
	
END_VAR

cntUpONS(CLK:= cntUp);
IF trackingEnable THEN
		IF cntUpONS.Q THEN
			count_index := count_index +1;
		END_IF
	FOR index :=0 TO NbMaxArrayDepth DO
		IF clr THEN
				count_index := 0;
				speedTracking[index].stateID:=-1;
				speedTracking[index].cycleArray:= speedTracking_mt;
		ELSIF  speedTracking[index].stateID = state THEN
			state_index := index;
			EXIT;
		ELSIF speedTracking[index].stateID = -1 THEN
			state_index := index;
			speedTracking[index].stateID := state;
			speedTracking[index].stateName := stateName;
			EXIT;
		END_IF
	END_FOR
	clr:=FALSE;
	stateTimer(PT:=T#10000S);
	IF state  = laststate THEN
		stateTimer.IN := TRUE;
	ELSIF state  <> laststate THEN
		stateTimer.IN := FALSE;
		laststate:=state;
	END_IF
IF stopTime> stateTimer.ET AND stateTimer.ET >T#0MS THEN
	speedTracking[state_index].cycleArray[count_index] := stateTimer.ET;
END_IF
	
	IF count_index >=20 THEN
		count_index :=0;
	END_IF
ELSE
	count_index := 0;
END_IF

END_FUNCTION_BLOCK

// Function Blocks/Electric Solenoid/FB_ElectricSolenoid
FUNCTION_BLOCK FB_ElectricSolenoid EXTENDS FB_BaseObject IMPLEMENTS ISimulateable, IUpDown
VAR_INPUT
	downFeedback : BOOL;
END_VAR
VAR_OUTPUT
	actuateSolenoid : BOOL;
END_VAR
VAR
	_simulateActive : BOOL;
END_VAR

END_FUNCTION_BLOCK

// Testing/Actuators/IUpDown
INTERFACE IUpDown EXTENDS IAllObjects

END_INTERFACE

// Function Blocks/IO/FB_IOLinkBlock
{attribute 'FBVisuCreator'}
FUNCTION_BLOCK FINAL FB_IOLinkBlock EXTENDS FB_Murr16PointCFGIO
VAR_INPUT
END_VAR
VAR_OUTPUT
	iIOLinkPort4 : WORD;
	iIOLinkPort5 : WORD;
	iIOLinkPort6 : WORD;
	iIOLinkPort7 : WORD;
END_VAR
VAR
END_VAR

SUPER^();

iIOLinkPort4 :=  TO_WORD(OSCAT_BASIC.WORD_OF_BYTE(B0 := ptrEIPInputs[3], B1 := ptrEIPInputs[2])); 
iIOLinkPort5 :=  TO_WORD(OSCAT_BASIC.WORD_OF_BYTE(B0 := ptrEIPInputs[5], B1 := ptrEIPInputs[4])); 
iIOLinkPort6 :=  TO_WORD(OSCAT_BASIC.WORD_OF_BYTE(B0 := ptrEIPInputs[7], B1 := ptrEIPInputs[6])); 
iIOLinkPort7 :=  TO_WORD(OSCAT_BASIC.WORD_OF_BYTE(B0 := ptrEIPInputs[9], B1 := ptrEIPInputs[8]));

END_FUNCTION_BLOCK

// Function Blocks/IO/FB_Murr16PointCFGIO
{attribute 'FBVisuCreator'}
FUNCTION_BLOCK FB_Murr16PointCFGIO EXTENDS FB_BaseObject 
VAR_INPUT
	ptrEIPInputs : POINTER TO BYTE;	// Pointer to starting word of EIP Inputs for the I/O Image
    ptrEIPOutputs : POINTER TO BYTE;	// Pointer to starting word of EIP Outputs for the I/O Image
	
	oPort0Pin2 : BOOL;
	oPort0Pin4 : BOOL;
	oPort1Pin2 : BOOL;
	oPort1Pin4 : BOOL;
	oPort2Pin2 : BOOL;
	oPort2Pin4 : BOOL;
	oPort3Pin2 : BOOL;
	oPort3Pin4 : BOOL;
	oPort4Pin2 : BOOL;
	oPort4Pin4 : BOOL;
	oPort5Pin2 : BOOL;
	oPort5Pin4 : BOOL;
	oPort6Pin2 : BOOL;
	oPort6Pin4 : BOOL;
	oPort7Pin2 : BOOL;
	oPort7Pin4 : BOOL;
END_VAR
VAR_OUTPUT
	iPort0Pin2 : BOOL;
	iPort0Pin4 : BOOL;
	iPort1Pin2 : BOOL;
	iPort1Pin4 : BOOL;
	iPort2Pin2 : BOOL;
	iPort2Pin4 : BOOL;
	iPort3Pin2 : BOOL;
	iPort3Pin4 : BOOL;
	iPort4Pin2 : BOOL;
	iPort4Pin4 : BOOL;
	iPort5Pin2 : BOOL;
	iPort5Pin4 : BOOL;
	iPort6Pin2 : BOOL;
	iPort6Pin4 : BOOL;
	iPort7Pin2 : BOOL;
	iPort7Pin4 : BOOL;
END_VAR
VAR_IN_OUT
END_VAR
VAR 
END_VAR


iPort0Pin2 := ptrEIPInputs[1].0;
iPort0Pin4 := ptrEIPInputs[0].0;
iPort1Pin2 := ptrEIPInputs[1].1;
iPort1Pin4 := ptrEIPInputs[0].1;
iPort2Pin2 := ptrEIPInputs[1].2;
iPort2Pin4 := ptrEIPInputs[0].2;
iPort3Pin2 := ptrEIPInputs[1].3;
iPort3Pin4 := ptrEIPInputs[0].3;
iPort4Pin2 := ptrEIPInputs[1].4;
iPort4Pin4 := ptrEIPInputs[0].4;
iPort5Pin2 := ptrEIPInputs[1].5;
iPort5Pin4 := ptrEIPInputs[0].5;
iPort6Pin2 := ptrEIPInputs[1].6;
iPort6Pin4 := ptrEIPInputs[0].6;
iPort7Pin2 := ptrEIPInputs[1].7;
iPort7Pin4 := ptrEIPInputs[0].7;

ptrEIPOutputs[1].0 := oPort0Pin2;
ptrEIPOutputs[0].0 := oPort0Pin4;
ptrEIPOutputs[1].1 := oPort1Pin2;
ptrEIPOutputs[0].1 := oPort1Pin4;
ptrEIPOutputs[1].2 := oPort2Pin2;
ptrEIPOutputs[0].2 := oPort2Pin4;
ptrEIPOutputs[1].3 := oPort3Pin2;
ptrEIPOutputs[0].3 := oPort3Pin4;
ptrEIPOutputs[1].4 := oPort4Pin2;
ptrEIPOutputs[0].4 := oPort4Pin4;
ptrEIPOutputs[1].5 := oPort5Pin2;
ptrEIPOutputs[0].5 := oPort5Pin4;
ptrEIPOutputs[1].6 := oPort6Pin2;
ptrEIPOutputs[0].6 := oPort6Pin4;
ptrEIPOutputs[1].7 := oPort7Pin2;
ptrEIPOutputs[0].7 := oPort7Pin4;

END_FUNCTION_BLOCK

// Function Blocks/IO/FB_Murr56691_IP20
{attribute 'FBVisuCreator'}
FUNCTION_BLOCK FB_Murr56691_IP20 EXTENDS FB_BaseObject 
VAR_INPUT
	ptrEIPInputs : POINTER TO BYTE;	// Pointer to starting word of EIP Inputs for the I/O Image
    ptrEIPOutputs : POINTER TO BYTE;	// Pointer to starting word of EIP Outputs for the I/O Image
	
	oX100 : BOOL;
	oX101 : BOOL;
	oX102 : BOOL;
	oX103 : BOOL;
	oX104 : BOOL;
	oX105 : BOOL;
	oX106 : BOOL;
	oX107 : BOOL;
END_VAR
VAR_OUTPUT
	
	iX000 : BOOL;
	iX001 : BOOL;
	iX002 : BOOL;
	iX003 : BOOL;
	iX004 : BOOL;
	iX005 : BOOL;
	iX006 : BOOL;
	iX007 : BOOL;

	iX100 : BOOL;
	iX101 : BOOL;
	iX102 : BOOL;
	iX103 : BOOL;
	iX104 : BOOL;
	iX105 : BOOL;
	iX106 : BOOL;
	iX107 : BOOL;
END_VAR
VAR_IN_OUT
END_VAR
VAR 
END_VAR

//	Function Block: FB_Murr56691_IP20
//	Description: Abstracts a Murr 56691 IP20 I/O Block
//	
//	Created by: Ben Hess
//	Created Date: Friday, October 19, 2018

iX100 := ptrEIPInputs[0].0;
iX101 := ptrEIPInputs[0].1;
iX102 := ptrEIPInputs[0].2;
iX103 := ptrEIPInputs[0].3;
iX104 := ptrEIPInputs[0].4;
iX105 := ptrEIPInputs[0].5;
iX106 := ptrEIPInputs[0].6;
iX107 := ptrEIPInputs[0].7;

iX000 := ptrEIPInputs[1].0;
iX001 := ptrEIPInputs[1].1;
iX002 := ptrEIPInputs[1].2;
iX003 := ptrEIPInputs[1].3;
iX004 := ptrEIPInputs[1].4;
iX005 := ptrEIPInputs[1].5;
iX006 := ptrEIPInputs[1].6;
iX007 := ptrEIPInputs[1].7;

ptrEIPOutputs[0].0 := oX100;
ptrEIPOutputs[0].1 := oX101;
ptrEIPOutputs[0].2 := oX102;
ptrEIPOutputs[0].3 := oX103;
ptrEIPOutputs[0].4 := oX104;
ptrEIPOutputs[0].5 := oX105;
ptrEIPOutputs[0].6 := oX106;
ptrEIPOutputs[0].7 := oX107;

END_FUNCTION_BLOCK

// Function Blocks/IO/FB_PhysicalAnalogInput
FUNCTION_BLOCK FB_PhysicalAnalogInput EXTENDS FB_BaseObject IMPLEMENTS IExecuteAutomatically, ILoggable
VAR_INPUT
	in : REFERENCE TO WORD;		// Raw Analog Input
	enableLogging : BOOL;		// Enable logging
	logDeadband : INT;			// Deadband to log changes
END_VAR
VAR_OUTPUT
	RawValue : WORD;
END_VAR
VAR
	logged : BOOL;
	loggedValue : INT;
END_VAR

END_FUNCTION_BLOCK

// Function Blocks/IO/FB_PhysicalDigitalOutput
FUNCTION_BLOCK FB_PhysicalDigitalOutput EXTENDS FB_BaseObject IMPLEMENTS ILoggable, ISimulateable
VAR_INPUT
	refOutput : REFERENCE TO BOOL; //  Reference to physical output
	
END_VAR
VAR_OUTPUT
	Q : BOOL;		// Logical inidcation of output
END_VAR
VAR
	outputONS : FB_ONS;
	_simulate : BOOL;	// Simulate output - do not trigger actual physical output
END_VAR
VAR_IN_OUT
	
END_VAR

END_FUNCTION_BLOCK

// Function Blocks/Machine Components/FB_MurrMaster
FUNCTION_BLOCK FB_MurrMaster EXTENDS FB_BaseObject
VAR_INPUT
	ptrEIPInputs : POINTER TO BYTE;	// Pointer to starting word of EIP Inputs for the I/O Image
    ptrEIPOutputs : POINTER TO BYTE;	// Pointer to starting word of EIP Outputs for the I/O Image
END_VAR
VAR_OUTPUT
	headIONode : FB_IOLinkBlock(name := 'Head Block');
	frontGuardIONode : FB_Murr16PointCFGIO(name := 'Front Guard Block');
	dischargeIONode : FB_Murr16PointCFGIO(name := 'Discharge Block');
	printerIONode : FB_Murr56691_IP20(name := 'Printer Block');
END_VAR
VAR
END_VAR
VAR (*Faults*)
	commFail : FB_Fault(name := CONCAT(_prefix,  'Communication Failure'));
END_VAR

// Head IO Node, offset of 0 for I/O
headIONode(ptrEIPInputs := ptrEIPInputs, ptrEIPOutputs := ptrEIPOutputs);
frontGuardIONode(ptrEIPInputs := ADR(ptrEIPInputs[30]), ptrEIPOutputs := ADR(ptrEIPOutputs[30]));
dischargeIONode(ptrEIPInputs := ADR(ptrEIPInputs[32]), ptrEIPOutputs := ADR(ptrEIPOutputs[32]));
printerIONode(ptrEIPInputs := ADR(ptrEIPInputs[34]), ptrEIPOutputs := ADR(ptrEIPOutputs[34]));
{region 'Alarms'}

{endregion}

END_FUNCTION_BLOCK

// Function Blocks/SolenoidValves/FB_DoubleSolenoidClosedCenterActuator
FUNCTION_BLOCK FB_DoubleSolenoidClosedCenterActuator EXTENDS FB_PneumaticActuator IMPLEMENTS IExtendLowPressure
VAR_INPUT
END_VAR
VAR_OUTPUT
END_VAR
VAR
	
END_VAR

END_FUNCTION_BLOCK

// Function Blocks/SolenoidValves/FB_PneumaticActuator
FUNCTION_BLOCK FB_PneumaticActuator EXTENDS FB_SolenoidValve IMPLEMENTS ICylinder
VAR_INPUT
END_VAR
VAR_OUTPUT
END_VAR
VAR
	_extendAsserted : BOOL;
	_isExtended : BOOL;
	_retractAsserted : BOOL;
	_isRetracted : BOOL;
END_VAR

END_FUNCTION_BLOCK

// Function Blocks/SolenoidValves/FB_SolenoidValve
FUNCTION_BLOCK FB_SolenoidValve EXTENDS FB_BaseObject IMPLEMENTS ISolenoidValve, ISimulateable
VAR_INPUT
END_VAR
VAR_OUTPUT
	solenoid0 : BOOL;
	solenoid1 : BOOL;
END_VAR
VAR
	_simulateActive : BOOL;
END_VAR

END_FUNCTION_BLOCK

// Testing/Actuators/ISolenoidValve
INTERFACE ISolenoidValve EXTENDS ISimulateable

END_INTERFACE

// Function Blocks/SolenoidValves/FB_DoubleSolenoidOpenCenterActuator
FUNCTION_BLOCK FINAL FB_DoubleSolenoidOpenCenterActuator EXTENDS FB_DoubleSolenoidClosedCenterActuator IMPLEMENTS IExhaustable
VAR_INPUT
END_VAR
VAR_OUTPUT
END_VAR
VAR
END_VAR

END_FUNCTION_BLOCK

// Function Blocks/SolenoidValves/FB_SingleSolenoidNormallyRetractedActuator
FUNCTION_BLOCK FB_SingleSolenoidNormallyRetractedActuator EXTENDS FB_PneumaticActuator IMPLEMENTS ICylinder
VAR_INPUT
END_VAR
VAR_OUTPUT
END_VAR
VAR
END_VAR

END_FUNCTION_BLOCK

// Function Blocks/SolenoidValves/FB_SolenoidValveManifold
FUNCTION_BLOCK FB_SolenoidValveManifold EXTENDS FB_BaseObject
VAR_INPUT
	ptrEIPOutputs : POINTER TO DWORD;	// Pointer to starting word of EIP Outputs for the I/O Image

	station : ARRAY[1..16] OF ISolenoidValve;	// Array of up to 16 valve stations on manifold 
	
END_VAR
VAR_OUTPUT
END_VAR
VAR
	i : INT;
	j : INT;
END_VAR

//	Function Block: FB_SolenoidValveManifold
//	Description: Sets the output image of the valve manifold (ptrEIPOutputs) to the correct values depending on configuration.  
//
//	Usage: All stations should be configured with a valve before running.
// 
//	Created by: Ben Hess
//	Created Date: 6-27-2019


// Loop through all possible stations
FOR i := 1 TO 16 DO
	IF station[i] <> 0 THEN	// Check for valid reference passed into the station interface
		// If ref good then set I/O image bit for proper station.  If simulated then don't set real output for solenoid
		ptrEIPOutputs^ := OSCAT_BASIC.BIT_LOAD_DW(in := ptrEIPOutputs^, POS := j, VAL := station[i].Solenoid0Asserted AND NOT station[i].Simulate);
		ptrEIPOutputs^ := OSCAT_BASIC.BIT_LOAD_DW(in := ptrEIPOutputs^, POS := j+1, VAL := station[i].Solenoid1Asserted AND NOT station[i].Simulate);
	END_IF
	j := j + 2;
END_FOR
// Restart bit loop
j := 0;

END_FUNCTION_BLOCK

// Function Blocks/SolenoidValves/FB_VacuumGenerator
FUNCTION_BLOCK FB_VacuumGenerator EXTENDS FB_SolenoidValve
VAR_INPUT
END_VAR
VAR_OUTPUT
END_VAR
VAR
END_VAR

END_FUNCTION_BLOCK

// Motion/Base/Axis_REF
{attribute 'FBVisuCreator'}
FUNCTION_BLOCK Axis_REF IMPLEMENTS IAxisRef
VAR_INPUT
	AxisState : AXIS_STATE;			// The axis state
	SetOpMode : OP_MODE; 			// The set opmode
	PowerOn : BOOL; 				// Regulator (power) on/off
	DriveEnable : BOOL;				// Deactivate (TRUE) or activate (FALSE) software halt/quickstop
	AckError : BOOL;				// Acknowledge error (fault reset)
	StartHoming : BOOL;				// Tells the axis to start homing, only used in homing mode
	Halt : BOOL; 					// Tells the axis to halt using a quick stop, used in all modes
	NewSetPoint : BOOL; 			// Tells the axis that a new set point has been given, only used in position mode
	MoveAbs : BOOL;					// Perform an absolute move
	MoveAbsTorque : BOOL;			// Perform an absolute move with a torque l
	MoveRel : BOOL;					// Perform a relative move
	MoveVelo : BOOL;				// Start a velocity move
	{attribute 'FBVisuCreatorFormatString' := '%1.2f'}
	TargetPosDist : REAL;			// The target position or distance in [u]
	{attribute 'FBVisuCreatorFormatString' := '%1.2f'}
	TargetVelocity : REAL;			// The target velocity in [u/s]
	{attribute 'FBVisuCreatorFormatString' := '%1.2f'}
	ProfileVelocity : REAL;			// The profile velocity in [u/s]
	{attribute 'FBVisuCreatorFormatString' := '%1.2f'}
	ProfileAcceleration : REAL;		// The profile acceleration in [u/s²]
	{attribute 'FBVisuCreatorFormatString' := '%1.2f'}
	ProfileDeceleration : REAL;		// The profile deceleration in [u/s²]
	{attribute 'FBVisuCreatorFormatString' := '%1.2f'}
	ProfileCurrentLimit : REAL;		// The profile current limit in [%]
	{attribute 'FBVisuCreatorFormatString' := '%1.2f'}
	QuickStopDeceleration : REAL;	// The deceleration for a quick stop in [u/s²]
	{attribute 'FBVisuCreatorFormatString' := '%1.2f'}
	DefaultCurrent : REAL;			// Default Current Limit [%]
END_VAR
VAR_OUTPUT
	{attribute 'FBVisuCreatorFormatString' := '%s'}
	ActOpMode : OP_MODE; 			// The actual opmode
	CommStatus : BOOL;				// Whether communication is OK
	PowerState : BOOL;				// Effective state of the power stage of the axis
	EnableState : BOOL;				// Effective state of the software halt/quickstop of the axis (TRUE: deactivated, FALSE: activated), 
	Error : BOOL; 					// Axis error
	{attribute 'FBVisuCreatorFormatString' := '%1.2f'}
	ActPos : REAL;					// Actual position in [u]
	{attribute 'FBVisuCreatorFormatString' := '%1.2f'}
	ActVelocity : REAL;				// Actual velocity in [u/s]
	SetPointAck : BOOL;				// Set if the new set point has been acknowledged, only used in position mode
	TargetReached : BOOL;			// Set if the target is reached, only set in position and homing mode
	InVelocity : BOOL; 				// Set if it has reached the commanded velocity, only set in velocity mode
	HomingDone : BOOL;				// Set if homing has been performed successfully (implies TargetReached), only set in homing mode
END_VAR
VAR
END_VAR
VAR_IN_OUT

END_VAR

END_FUNCTION_BLOCK

// Motion/Base/IAxisRef
INTERFACE IAxisRef EXTENDS __System.IQueryInterface

END_INTERFACE

// Motion/Base/MC_Base
FUNCTION_BLOCK MC_Base
VAR_INPUT
	Execute : BOOL; 		// Rising edge: The halt is started 
END_VAR
VAR_OUTPUT
	Done : BOOL;			// Becomes true as soon as the axis has reached velocity zero
	Busy : BOOL;			// TRUE as long as MC_Halt is operating, reset when velocity is zero
	CommandAborted : BOOL;	// Commanded motion was interrupted by any motion FB acting on the same axis
	Error : BOOL;			// Signals that an error has occured
	ErrorID : MC_ERROR;		// Error number
END_VAR
VAR
	ExecuteOSR : Standard.R_TRIG;
	ExecuteOSF : Standard.F_TRIG;
	MC_State : INT;
END_VAR
VAR_IN_OUT
	Axis : Axis_REF;		// Reference to the axis 
END_VAR

END_FUNCTION_BLOCK

// Motion/PLCopen MC/MC_Halt
FUNCTION_BLOCK FINAL MC_Halt EXTENDS MC_Base
VAR_INPUT
	Deceleration : REAL; 	// Value of the deceleration (decreasing energy of the motor) [u/s²]
END_VAR
VAR_OUTPUT
END_VAR
VAR
END_VAR

//	Function Block: MC_Halt
//	Description: Commands a controlled motion stop. The axis is moved to the state DiscreteMotion, until the velocity is zero. 
//				 When the output Done is set, the state is transferred to Standstill.
//	Created by: Ben Hess
//	Created Date: May 3rd, 2019

ExecuteOSR(CLK := Execute);

IF MC_State <> 0 AND Axis.Error THEN
	SetError();
	ErrorID := MC_ERROR.AXIS_ERROR_DURING_COMMAND;
	MC_State := 0;
	Axis.Halt := FALSE;
	Axis.AxisState := AXIS_STATE.AS_Standstill;
END_IF

CASE MC_State OF
	0:		// Idle State.  If execute rising edge then start halt 
			IF ExecuteOSR.Q THEN
				IF NOT Axis.Error AND Axis.PowerState THEN
					SetBusy();
					Axis.AxisState := AXIS_STATE.AS_DiscreteMotion;
					Axis.QuickStopDeceleration := Deceleration;
					Axis.Halt := TRUE;
					MC_State := 1;
				ELSE
					Error := TRUE;
					ErrorID := MC_ERROR.AXIS_NOT_READY;
				END_IF
				
			END_IF
	
	1:		// Stopping.  Once stopped go back to idle
			IF Axis.ActVelocity = 0 THEN
				Axis.Halt := FALSE;
				Axis.AxisState := AXIS_STATE.AS_Standstill;
				SetDone();
				MC_State := 0;
			END_IF
			
	99: 		// Error
END_CASE

END_FUNCTION_BLOCK

// Motion/Custom MC/MC_MoveAbsoluteTorqueLimited
FUNCTION_BLOCK MC_MoveAbsoluteTorqueLimited EXTENDS MC_Base
VAR_INPUT
	Position : REAL;		// Commanded position for the motion (may be negative) (in technical units [u])
	Velocity : REAL;		// Value of the maximum velocity (always positive) (not necessarily reached) [u/s]
	Acceleration : REAL;	// Value of the acceleration (always positive) (increasing energy of the motor) [u/s²]
	Deceleration : REAL;	// Value of the deceleration (always positive) (decreasing energy of the motor) [u/s²]
	CurrentLimit : REAL;	// Maximum current allowed to perform the move [A]
END_VAR
VAR_OUTPUT
END_VAR
VAR
END_VAR

//	Function Block: MC_MoveAbsoluteTorqueLimited
//	Description: Commands a controlled motion to a specified absolute position with torque limiting.
//				 After completion, the axis state is Standstill.
//				 This FB is an extention of the PLCOpen standard
//	Created by: Ben Hess
//	Created Date: May 3rd, 2019

ExecuteOSR(CLK := Execute);
ExecuteOSF(CLK := Execute);

IF MC_State <> 0 AND Axis.Error THEN
	SetError();
	ErrorID := MC_ERROR.AXIS_ERROR_DURING_COMMAND;
	MC_State := 0;
	Axis.MoveAbsTorque := FALSE;
END_IF


CASE MC_State OF
	0:		// Idle State.  If execute rising edge then start absolute move 
			IF ExecuteOSR.Q THEN
				IF NOT Axis.Error AND Axis.PowerState THEN
					SetBusy();
					Axis.TargetPosDist := Position;
					Axis.ProfileVelocity := Velocity;
					Axis.ProfileAcceleration := Acceleration;
					Axis.ProfileDeceleration := Deceleration;
					Axis.ProfileCurrentLimit := CurrentLimit;
					Axis.MoveAbsTorque := TRUE;
					MC_State := 1;
				ELSE
					SetError();
					ErrorID := MC_ERROR.AXIS_NOT_READY;
				END_IF
			END_IF
	
	1:		// Wait for target reached.  Once stopped go back to idle
			IF Axis.TargetReached THEN
				Axis.MoveAbsTorque := FALSE;
				SetDone();
				MC_State := 0;
			ELSIF Axis.AxisState <> AXIS_STATE.AS_DiscreteMotion THEN
				Axis.MoveAbsTorque := FALSE;
				SetError();
				MC_State := 0;
			END_IF
END_CASE

END_FUNCTION_BLOCK

// Motion/Custom MC/MC_MoveFinalBagDelivery
FUNCTION_BLOCK MC_MoveFinalBagDelivery EXTENDS MC_MoveAbsolute
VAR_INPUT
	Position : REAL;		// Commanded position for the motion (may be negative) (in technical units [u])
	Velocity : REAL;		// Value of the maximum velocity (always positive) (not necessarily reached) [u/s]
	Acceleration : REAL;	// Value of the acceleration (always positive) (increasing energy of the motor) [u/s²]
	Deceleration : REAL;	// Value of the deceleration (always positive) (decreasing energy of the motor) [u/s²]
END_VAR
VAR_OUTPUT
END_VAR
VAR
END_VAR

//	Function Block: MC_MoveFinalBagDelivery
//	Description: Commands a controlled motion to a specified absolute position.
//				 After completion, the axis state is Standstill.
//	Created by: Ben Hess
//	Created Date: July 1st, 2019

ExecuteOSR(CLK := Execute);
ExecuteOSF(CLK := Execute);

IF MC_State <> 0 AND Axis.Error THEN
	SetError();
	ErrorID := MC_ERROR.AXIS_ERROR_DURING_COMMAND;
	MC_State := 0;
	Axis.MoveAbs := FALSE;
END_IF


CASE MC_State OF
	0:		// Idle State.  If execute rising edge then start absolute move 
			IF ExecuteOSR.Q THEN
				IF NOT Axis.Error AND Axis.PowerState THEN
					SetBusy();
					Axis.TargetPosDist := Position;
					Axis.ProfileVelocity := Velocity;
					Axis.ProfileAcceleration := Acceleration;
					Axis.ProfileDeceleration := Deceleration;
					Axis.MoveAbs := TRUE;
					MC_State := 1;
				ELSE
					SetError();
					ErrorID := MC_ERROR.AXIS_NOT_READY;
				END_IF
			END_IF
	
	1:		// Wait for target reached.  Once stopped go back to idle
			IF Axis.TargetReached THEN
				Axis.MoveAbs := FALSE;
				SetDone();
				MC_State := 0;
			ELSIF Axis.AxisState <> AXIS_STATE.AS_DiscreteMotion THEN
				Axis.MoveAbs := FALSE;
				SetAborted();
				MC_State := 0;
			END_IF
END_CASE

END_FUNCTION_BLOCK

// Motion/PLCopen MC/MC_MoveAbsolute
FUNCTION_BLOCK MC_MoveAbsolute EXTENDS MC_Base
VAR_INPUT
	Position : REAL;		// Commanded position for the motion (may be negative) (in technical units [u])
	Velocity : REAL;		// Value of the maximum velocity (always positive) (not necessarily reached) [u/s]
	Acceleration : REAL;	// Value of the acceleration (always positive) (increasing energy of the motor) [u/s²]
	Deceleration : REAL;	// Value of the deceleration (always positive) (decreasing energy of the motor) [u/s²]
END_VAR
VAR_OUTPUT
END_VAR
VAR
END_VAR

//	Function Block: MC_MoveAbsolute
//	Description: Commands a controlled motion to a specified absolute position.
//				 After completion, the axis state is Standstill.
//	Created by: Ben Hess
//	Created Date: May 3rd, 2019

ExecuteOSR(CLK := Execute);
ExecuteOSF(CLK := Execute);

IF MC_State <> 0 AND Axis.Error THEN
	SetError();
	ErrorID := MC_ERROR.AXIS_ERROR_DURING_COMMAND;
	MC_State := 0;
	Axis.MoveAbs := FALSE;
END_IF


CASE MC_State OF
	0:		// Idle State.  If execute rising edge then start absolute move 
			IF ExecuteOSR.Q THEN
				IF NOT Axis.Error AND Axis.PowerState THEN
					SetBusy();
					Axis.AxisState := AXIS_STATE.AS_DiscreteMotion;
					Axis.TargetPosDist := Position;
					Axis.ProfileVelocity := Velocity;
					Axis.ProfileAcceleration := Acceleration;
					Axis.ProfileDeceleration := Deceleration;
					Axis.ProfileCurrentLimit := Axis.DefaultCurrent;
					Axis.MoveAbs := TRUE;
					MC_State := 1;
					ErrorID := MC_ERROR.NO_ERROR;
				ELSE
					SetError();
					ErrorID := MC_ERROR.AXIS_NOT_READY;
				END_IF
			END_IF
	
	1:		// Wait for target reached.  Once stopped go back to idle
			IF Axis.TargetReached THEN
				Axis.MoveAbs := FALSE;
				SetDone();
				MC_State := 0;
			ELSIF Axis.AxisState <> AXIS_STATE.AS_DiscreteMotion OR CommandAborted THEN
				Axis.MoveAbs := FALSE;
				SetAborted();
				MC_State := 0;
			END_IF
END_CASE

END_FUNCTION_BLOCK

// Motion/PLCopen MC/MC_Home
FUNCTION_BLOCK FINAL MC_Home EXTENDS MC_Base
VAR_INPUT
END_VAR
VAR_OUTPUT
END_VAR
VAR

END_VAR

//	Function Block: MC_Home
//	Description: Commands the axis to perform the «search home» sequence. The details of this sequence are manufacturer specific and can be set by the axis’ parameters. 
//				 After completion, the axis state is Standstill if it was Standstill when started.
//	Created by: Ben Hess
//	Created Date: May 3rd, 2019

ExecuteOSR(CLK := Execute);

IF MC_State <> 0 AND Axis.Error THEN
	SetError();
	ErrorID := MC_ERROR.AXIS_ERROR_DURING_COMMAND;
	MC_State := 0;
	Axis.StartHoming := FALSE;
	Axis.AxisState := AXIS_STATE.AS_Standstill;
END_IF


CASE MC_State OF
	0:		// Idle State.  If execute rising edge then start halt 
			IF ExecuteOSR.Q THEN
				IF NOT Axis.Error AND Axis.PowerState THEN
					SetBusy();
					Axis.AxisState := AXIS_STATE.AS_Homing;
					Axis.StartHoming := TRUE;
					MC_State := 1;
				ELSE
					Error := TRUE;
					ErrorID := MC_ERROR.AXIS_NOT_READY;
				END_IF
				
			END_IF
	
	1:		// Stopping.  Once stopped go back to idle
			IF Axis.HomingDone THEN
				Axis.StartHoming := FALSE;
				Axis.AxisState := AXIS_STATE.AS_Standstill;
				SetDone();
				MC_State := 0;
			END_IF
END_CASE

END_FUNCTION_BLOCK

// Motion/PLCopen MC/MC_MoveRelative
FUNCTION_BLOCK MC_MoveRelative EXTENDS MC_Base
VAR_INPUT
	Distance : REAL;		// Relative distance for the motion (in technical units [u])
	Velocity : REAL;		// Value of the maximum velocity (always positive) (not necessarily reached) [u/s]
	Acceleration : REAL;	// Value of the acceleration (always positive) (increasing energy of the motor) [u/s²]
	Deceleration : REAL;	// Value of the deceleration (always positive) (decreasing energy of the motor) [u/s²]
END_VAR
VAR_OUTPUT
END_VAR
VAR
END_VAR

//	Function Block: MC_MoveRelative
//	Description: Commands a controlled motion of a specified distance relative to the position at the time of the execution.
//				 The motion completes with velocity zero.
//				 After completion, the axis state is Standstill.
//	Created by: Ben Hess
//	Created Date: May 6th, 2019

ExecuteOSR(CLK := Execute);

IF MC_State <> 0 AND Axis.Error THEN
	SetError();
	ErrorID := MC_ERROR.AXIS_ERROR_DURING_COMMAND;
	MC_State := 0;
	Axis.MoveRel := FALSE;
	Axis.AxisState := AXIS_STATE.AS_ErrorStop;
END_IF


CASE MC_State OF
	0:		// Idle State.  If execute rising edge then start absolute move 
			IF ExecuteOSR.Q THEN
				IF NOT Axis.Error AND Axis.PowerState THEN
					SetBusy();
					Axis.AxisState := AXIS_STATE.AS_DiscreteMotion;
					Axis.TargetPosDist := Distance;
					Axis.ProfileVelocity := Velocity;
					Axis.ProfileAcceleration := Acceleration;
					Axis.ProfileDeceleration := Deceleration;
					Axis.ProfileCurrentLimit := Axis.DefaultCurrent;
					Axis.MoveRel := TRUE;
					MC_State := 1;
					ErrorID := MC_ERROR.NO_ERROR;
				ELSE
					Error := TRUE;
					ErrorID := MC_ERROR.AXIS_NOT_READY;
				END_IF
			END_IF
	
	1:		// Wait for target reached.  Once stopped go back to idle
			IF Axis.TargetReached THEN
				Axis.MoveRel := FALSE;
				Axis.AxisState := AXIS_STATE.AS_Standstill;
				SetDone();
				MC_State := 0;
			ELSIF Axis.AxisState <> AXIS_STATE.AS_DiscreteMotion OR CommandAborted OR NOT Execute THEN
				Axis.MoveRel := FALSE;
				SetAborted();
				MC_State := 0;
			END_IF
END_CASE

END_FUNCTION_BLOCK

// Motion/PLCopen MC/MC_MoveVelocity
FUNCTION_BLOCK MC_MoveVelocity
VAR_INPUT
	Execute : BOOL; 		// Rising edge: The halt is started 
	Velocity : REAL;		// Value of the maximum velocity (always positive) (not necessarily reached) [u/s]
	Acceleration : REAL;	// Value of the acceleration (always positive) (increasing energy of the motor) [u/s²]
	Deceleration : REAL;	// Value of the deceleration (always positive) (decreasing energy of the motor) [u/s²]
END_VAR
VAR_OUTPUT
	InVelocity : BOOL;		// Value of the commanded velocity (may be negative) (not necessarily reached) [u/s]
	Busy : BOOL;			// TRUE as long as MC_Halt is operating, reset when velocity is zero
	CommandAborted : BOOL;	// Commanded motion was interrupted by any motion FB acting on the same axis
	Error : BOOL;			// Signals that an error has occured
	ErrorID : MC_ERROR;		// Error number
END_VAR
VAR
	ExecuteOSR : Standard.R_TRIG;
	MC_State : INT;
END_VAR
VAR_IN_OUT
	Axis : Axis_REF;		// Reference to the axis 
END_VAR

//	Function Block: MC_MoveVelocity
//	Description: Commands a never ending controlled motion with a specified velocity.
//				 To stop the motion, the motion has to be interrupted by another motion command.
//				 The output InVelocity is reset when the block is aborted by another block.
//	Created by: Ben Hess
//	Created Date: May 6th, 2019

ExecuteOSR(CLK := Execute);

IF MC_State <> 0 AND Axis.Error THEN
	SetError();
	ErrorID := MC_ERROR.AXIS_ERROR_DURING_COMMAND;
	MC_State := 0;
	Axis.MoveVelo := FALSE;
	Axis.AxisState := AXIS_STATE.AS_ErrorStop;
END_IF


CASE MC_State OF
	0:		// Idle State.  If execute rising edge then start absolute move 
			IF ExecuteOSR.Q THEN
				IF NOT Axis.Error AND Axis.PowerState THEN
					SetBusy();
					Axis.AxisState := AXIS_STATE.AS_ContinuousMotion;
					Axis.ProfileVelocity := Velocity;
					Axis.ProfileAcceleration := Acceleration;
					Axis.ProfileDeceleration := Deceleration;
					Axis.ProfileCurrentLimit := Axis.DefaultCurrent;
					Axis.MoveVelo := TRUE;
					MC_State := 1;
				ELSE
					Error := TRUE;
					ErrorID := MC_ERROR.AXIS_NOT_READY;
				END_IF
			END_IF
	
	1:		// Wait for target reached.
			IF Axis.InVelocity THEN
				Axis.MoveVelo := FALSE;
				SetInVelo();
				MC_State := 2;
			END_IF
	
	2:		// If another MC turns off velocity mode then go back to idle
			IF NOT Axis.InVelocity THEN
				InVelocity := FALSE;
				MC_State := 0;
			END_IF
END_CASE

END_FUNCTION_BLOCK

// Motion/PLCopen MC/MC_Power
FUNCTION_BLOCK MC_Power
VAR_INPUT
	Enable : BOOL; 			// Enables the FUNCTION block 
	RegulatorOn : BOOL; 	// Enables the power stage 
	DriveStart : BOOL; 		// Disables the quickstop mechanism 
END_VAR
VAR_OUTPUT
	Status : BOOL; 					// Axis ready for motion 
	RegulatorRealState : BOOL; 		// Effective state OF the power stage 
	DriveStartRealState : BOOL; 	// Effective state of the quickstop mechanism 
	Busy : BOOL; 					// Function block is executing 
	Error : BOOL; 					// Signals that an error has occured 
	ErrorID : MC_ERROR; 			// Error number 
END_VAR
VAR
	EnableOSR : Standard.R_TRIG;
	MC_State : INT;
END_VAR
VAR_IN_OUT
	Axis : Axis_REF;		// Reference to the axis 
END_VAR

//	Function Block: MC_Power
//	Description: 	Controls the power stage of an axis and can be used to issue a quick stop.
//					◾A call of MC_Power_SML with bRegulatorOn=FALSE sets the axis state to PowerOff (disabled).
//					◾A call of MC_Power_SML with bRegulatorOn``=``TRUE on a disabled axis sets the axis state to Standstill, if there is no error on the axis. If an error is detected, the state of the axis is set to ErrorStop.
//					◾If the inputs Enable, bRegulatorOn and bDriveStart are ``TRUE but the output Status remains in FALSE for a long time, there may be a problem with the power stage, or an external halt may be set.
//					◾If power fails (also during operation), the axis state is set to ErrorStop.
//	Created by: Ben Hess
//	Created Date: May 6th, 2019

Status := Axis.PowerState AND Axis.EnableState;

RegulatorRealState := Axis.PowerState;
DriveStartRealState := Axis.EnableState;

IF NOT Enable THEN
	Axis.PowerOn := Axis.DriveEnable := FALSE;
ELSE
	Axis.PowerOn := RegulatorOn;
	Axis.DriveEnable := DriveStart;
END_IF

END_FUNCTION_BLOCK

// Motion/PLCopen MC/MC_Reset
FUNCTION_BLOCK FINAL MC_Reset EXTENDS MC_Base
VAR_INPUT
END_VAR
VAR_OUTPUT
END_VAR
VAR

END_VAR

//	Function Block: MC_Reset
//	Description: Forces the transition from the state ErrorStop to Standstill or PowerOff by resetting all internal axis-related errors.
//				 If the axis is not in state ErrorStop, the function block signals the error R_NO_ERROR_TO_RESET.
//	Created by: Ben Hess
//	Created Date: May 14th, 2019

ExecuteOSR(CLK := Execute);

IF MC_State <> 0 AND Axis.Error THEN
	SetError();
	ErrorID := MC_ERROR.AXIS_ERROR_DURING_COMMAND;
	MC_State := 0;
	Axis.AckError := FALSE;
END_IF


CASE MC_State OF
	0:		// Idle State.  If execute rising edge then start halt 
			IF ExecuteOSR.Q THEN
				//IF Axis.Error THEN
					SetBusy();
					Axis.AckError := TRUE;
					MC_State := 1;
				//ELSE
				//	Error := TRUE;
				//	ErrorID := MC_ERROR.R_NO_ERROR_TO_RESET;
				//END_IF
			END_IF
	
	1:		// Clearing error.  Once stopped go back to idle
			IF NOT Axis.Error THEN
				Axis.AckError := FALSE;
				Axis.AxisState := AXIS_STATE.AS_Standstill;
				SetDone();
				MC_State := 0;
			END_IF
END_CASE

END_FUNCTION_BLOCK

// Motion/PLCopen MC/MC_Stop
FUNCTION_BLOCK FINAL MC_Stop EXTENDS MC_Base
VAR_INPUT
	Deceleration : REAL; 	// Value of the deceleration (decreasing energy of the motor) [u/s²]
END_VAR
VAR_OUTPUT
END_VAR
VAR
END_VAR

//	Function Block: MC_Stop
//	Description: 	Executes a (blocking) stop on the axis.
//					As long as the Execute input is set or the stop is not finished, no other motion command is possible on the axis, 
//					and the axis state is Stopping. After both the stop is finished and Execute is reset, the axis status is set to Standstill.

//	Created by: Ben Hess
//	Created Date: May 3rd, 2019

ExecuteOSR(CLK := Execute);

IF MC_State <> 0 AND Axis.Error THEN
	SetError();
	ErrorID := MC_ERROR.AXIS_ERROR_DURING_COMMAND;
	MC_State := 0;
	Axis.Halt := FALSE;
	Axis.AxisState := AXIS_STATE.AS_Standstill;
END_IF

CASE MC_State OF
	0:		// Idle State.  If execute rising edge then start halt 
			IF ExecuteOSR.Q THEN
				IF NOT Axis.Error AND Axis.PowerState THEN
					SetBusy();
					Axis.AxisState := AXIS_STATE.AS_DiscreteMotion;
					Axis.QuickStopDeceleration := Deceleration;
					Axis.Halt := TRUE;
					MC_State := 1;
				ELSE
					Error := TRUE;
					ErrorID := MC_ERROR.AXIS_NOT_READY;
				END_IF
				
			END_IF
	
	1:		// Stopping.  Once stopped go back to idle
			IF Axis.ActVelocity = 0 THEN
				Axis.Halt := FALSE;
				Axis.AxisState := AXIS_STATE.AS_Standstill;
				SetDone();
				MC_State := 0;
			END_IF
			
	99: 		// Error
END_CASE

END_FUNCTION_BLOCK

// Testing/Actuators/FB_DummyUpDown
FUNCTION_BLOCK FB_DummyUpDown IMPLEMENTS IUpDown
VAR_INPUT
END_VAR
VAR_OUTPUT
END_VAR
VAR
END_VAR

END_FUNCTION_BLOCK

// Testing/Actuators/FB_PneumaticVerticalActuator
FUNCTION_BLOCK FB_PneumaticVerticalActuator EXTENDS FB_PneumaticActuator IMPLEMENTS IUpDown
VAR_INPUT
	cylinder : ICylinder;
END_VAR
VAR_OUTPUT
END_VAR
VAR
END_VAR
VAR_IN_OUT	
END_VAR

//	Function Block: FB_PneumaticVerticalActuator
//	Description: Wrapper for a cylinder with Up/Down substitiuted for Extend/Retract
//				  
//
//	Usage: 
// 
//	Created by: Ben Hess
//	Created Date: 6-27-2019

EnableSimulation(cylinder, _simulateActive);

END_FUNCTION_BLOCK

// Testing/HelperFunctions/EnableSimulation
FUNCTION EnableSimulation : BOOL
VAR_INPUT
	device : IAllObjects;
	enableSim : BOOL;
END_VAR
VAR
	simulatable : ISimulateable;
END_VAR

//	Function: EnableSimulation()
//	Description: Helper function
//				 Pass in a device. Set simulation status if possible
//	Created by: Ben Hess
//	Created Date: June 25th, 2019

IF (__QUERYINTERFACE(device, simulatable)) THEN
	simulatable.Simulate := enableSim;
END_IF

END_FUNCTION

// Testing/FB_AMPMotorSerial/FB_AMPMotorSerial
FUNCTION_BLOCK FB_AMPMotorSerial EXTENDS CBM.ETrig
VAR_INPUT
	sendData : STRING[60];
	inputs : POINTER TO BYTE;
	outputs : POINTER TO BYTE;
END_VAR
VAR_OUTPUT
	receivedData : STRING[60];
END_VAR
VAR
	serialState : eSerialStates;
	executeONS : FB_ONS;
	readBufferHasData : BOOL;
	readBufferDataSize : BYTE;
	writeBufferDataSize : BYTE;
	readTimeout : Standard.TON := (PT := T#30MS);
	timeToResponse : TIME;
	TA : BOOL;
	TR : BOOL;
	RA : BOOL;
	RR : BOOL;
	ClearOutReadBuffer : BOOL;
END_VAR
VAR_IN_OUT

END_VAR

executeONS(CLK := xExecute);
RR := inputs[0].2;
TA := inputs[0].1;

IF executeONS.OSF THEN
	serialState := eSerialStates.Idle;
END_IF
readBufferHasData := inputs[0].4;
readBufferDataSize := inputs[1];
readTimeout(IN := serialState = eSerialStates.getResponse); 

// IF readBufferHasData AND serialState = eSerialStates.Idle THEN
// 	ClearOutReadBuffer := TRUE;
// ELSE 
// 	ClearOutReadBuffer := FALSE;
// END_IF

CASE serialState OF
	eSerialStates.Idle :				// Wait for execute
										IF NOT xExecute THEN 
											xDone := FALSE;
											xBusy := FALSE;
										END_IF
										IF executeONS.OSR THEN
											xDone := FALSE;
											OSCAT_BASIC._STRING_TO_BUFFER(STR := sendData,0,ADR(outputs[2]),TO_UINT(LEN(sendData)));
											outputs[1] := TO_BYTE(Standard.LEN(sendData));
											IF TA THEN
												TR := FALSE;
											ELSE
												TR := TRUE;
											END_IF
											xBusy := TRUE;
											serialState := eSerialStates.writingOutBuffer;
										END_IF
	
	eSerialStates.writeOutBuffer :		// 
										
	
	eSerialStates.writingOutBuffer :	// 
										IF TA = TR THEN
											serialState := eSerialStates.getResponse;
										END_IF
	
	eSerialStates.getResponse :			//
										IF readBufferHasData THEN
											IF readTimeout.Q THEN
												timeToResponse := readTimeout.ET;
												IF RR THEN
													RA := FALSE;
												ELSE
													RA := TRUE;
												END_IF
												serialState := eSerialStates.gettingResponse;
											END_IF
											
										ELSIF readTimeout.Q THEN
											receivedData := '';
											xDone := TRUE;
											xBusy := FALSE;
											serialState := eSerialStates.Idle;
										END_IF
	
	eSerialStates.gettingResponse:		IF RA = RR THEN
											receivedData := OSCAT_BASIC.BUFFER_TO_STRING(PT := ADR(inputs[2]),SIZE := 50, 0, readBufferDataSize + 1);
											xDone := TRUE;
											xBusy := FALSE;
											serialState := eSerialStates.Idle;
										END_IF

	
END_CASE
//outputs[0].0 := ClearOutReadBuffer;
outputs[0].1 := TR;
outputs[0].2 := RA;

END_FUNCTION_BLOCK

// Testing/FB_BannerPalmButton/FB_BannerPalmButton
FUNCTION_BLOCK FB_BannerPalmButton
VAR_INPUT
	baggerReady : BOOL;
	baggerFaulted : BOOL;
	baggerInCycle : BOOL;
END_VAR
VAR_OUTPUT
	palmState0Output : BOOL;
	palmState1Output : BOOL;
END_VAR
VAR
END_VAR

palmState0Output := FALSE;
palmState1Output := FALSE;
IF baggerReady THEN
	palmState0Output := TRUE;
	palmState1Output := FALSE;
END_IF
IF baggerInCycle THEN
	palmState0Output := TRUE;
	palmState1Output := TRUE;
END_IF
IF baggerFaulted THEN
	palmState0Output := FALSE;
	palmState1Output := TRUE;
END_IF

END_FUNCTION_BLOCK

// Testing/FB_CrevisSerial/FB_CrevisSerial
FUNCTION_BLOCK FB_CrevisSerial EXTENDS CBM.ETrig
VAR_INPUT
	sendData : STRING[60];
	inputs : POINTER TO BYTE;
	outputs : POINTER TO BYTE;
END_VAR
VAR_OUTPUT
	receivedData : STRING[60];
END_VAR
VAR
	serialState : eSerialStates;
	executeONS : FB_ONS;
	readBufferHasData : BOOL;
	readBufferDataSize : BYTE;
	writeBufferDataSize : BYTE;
	readTimeout : Standard.TON := (PT := T#30MS);
	timeToResponse : TIME;
	TA : BOOL;
	TR : BOOL;
	RA : BOOL;
	RR : BOOL;
	ClearOutReadBuffer : BOOL;
END_VAR
VAR_IN_OUT

END_VAR

executeONS(CLK := xExecute);
RR := inputs[0].2;
TA := inputs[0].1;

IF executeONS.OSF THEN
	serialState := eSerialStates.Idle;
END_IF
readBufferHasData := inputs[0].4;
readBufferDataSize := inputs[1];
readTimeout(IN := serialState = eSerialStates.getResponse); 

// IF readBufferHasData AND serialState = eSerialStates.Idle THEN
// 	ClearOutReadBuffer := TRUE;
// ELSE 
// 	ClearOutReadBuffer := FALSE;
// END_IF

CASE serialState OF
	eSerialStates.Idle :				// Wait for execute
										IF NOT xExecute THEN 
											xDone := FALSE;
										END_IF
										IF executeONS.OSR THEN
											xDone := FALSE;
											OSCAT_BASIC._STRING_TO_BUFFER(STR := sendData,0,ADR(outputs[2]),TO_UINT(LEN(sendData)));
											outputs[1] := TO_BYTE(Standard.LEN(sendData));
											IF TA THEN
												TR := FALSE;
											ELSE
												TR := TRUE;
											END_IF
											xBusy := TRUE;
											serialState := eSerialStates.writingOutBuffer;
										END_IF
	
	eSerialStates.writeOutBuffer :		// 
										
	
	eSerialStates.writingOutBuffer :	// 
										IF TA = TR THEN
											serialState := eSerialStates.getResponse;
										END_IF
	
	eSerialStates.getResponse :			//
										IF readBufferHasData THEN
											IF readTimeout.Q THEN
												timeToResponse := readTimeout.ET;
												IF RR THEN
													RA := FALSE;
												ELSE
													RA := TRUE;
												END_IF
												serialState := eSerialStates.gettingResponse;
											END_IF
											
										ELSIF readTimeout.Q THEN
											receivedData := '';
											xDone := TRUE;
											xBusy := FALSE;
											serialState := eSerialStates.Idle;
										END_IF
	
	eSerialStates.gettingResponse:		IF RA = RR THEN
											receivedData := OSCAT_BASIC.BUFFER_TO_STRING(PT := ADR(inputs[2]),SIZE := 50, 0, readBufferDataSize + 1);
											xDone := TRUE;
											xBusy := FALSE;
											serialState := eSerialStates.Idle;
										END_IF

	
END_CASE
//outputs[0].0 := ClearOutReadBuffer;
outputs[0].1 := TR;
outputs[0].2 := RA;

END_FUNCTION_BLOCK

// Testing/HelperFunctions/ExhaustIfPossible
FUNCTION ExhaustIfPossible : BOOL  // Attempts to exhaust SV, returns true if exhaust commanded
VAR_INPUT
	device : IAllObjects;
END_VAR
VAR
	exhaustableDevice : IExhaustable;
END_VAR

//	Function: ExhaustIfPossible()
//	Description: Helper function
//				 Pass in a device that is controlled byt a SV - exhaust if possible
//	Created by: Ben Hess
//	Created Date: June 25th, 2019

IF (__QUERYINTERFACE(device, exhaustableDevice)) THEN
	exhaustableDevice.Exhaust();
	ExhaustIfPossible := TRUE;
ELSE
	ExhaustIfPossible := FALSE;
END_IF

END_FUNCTION

// Testing/HelperFunctions/ExtendLPIfPossible
FUNCTION ExtendLPIfPossible : BOOL
VAR_INPUT
	device : IAllObjects;
END_VAR
VAR
	extendLowPressureDevice : IExtendLowPressure;
END_VAR

